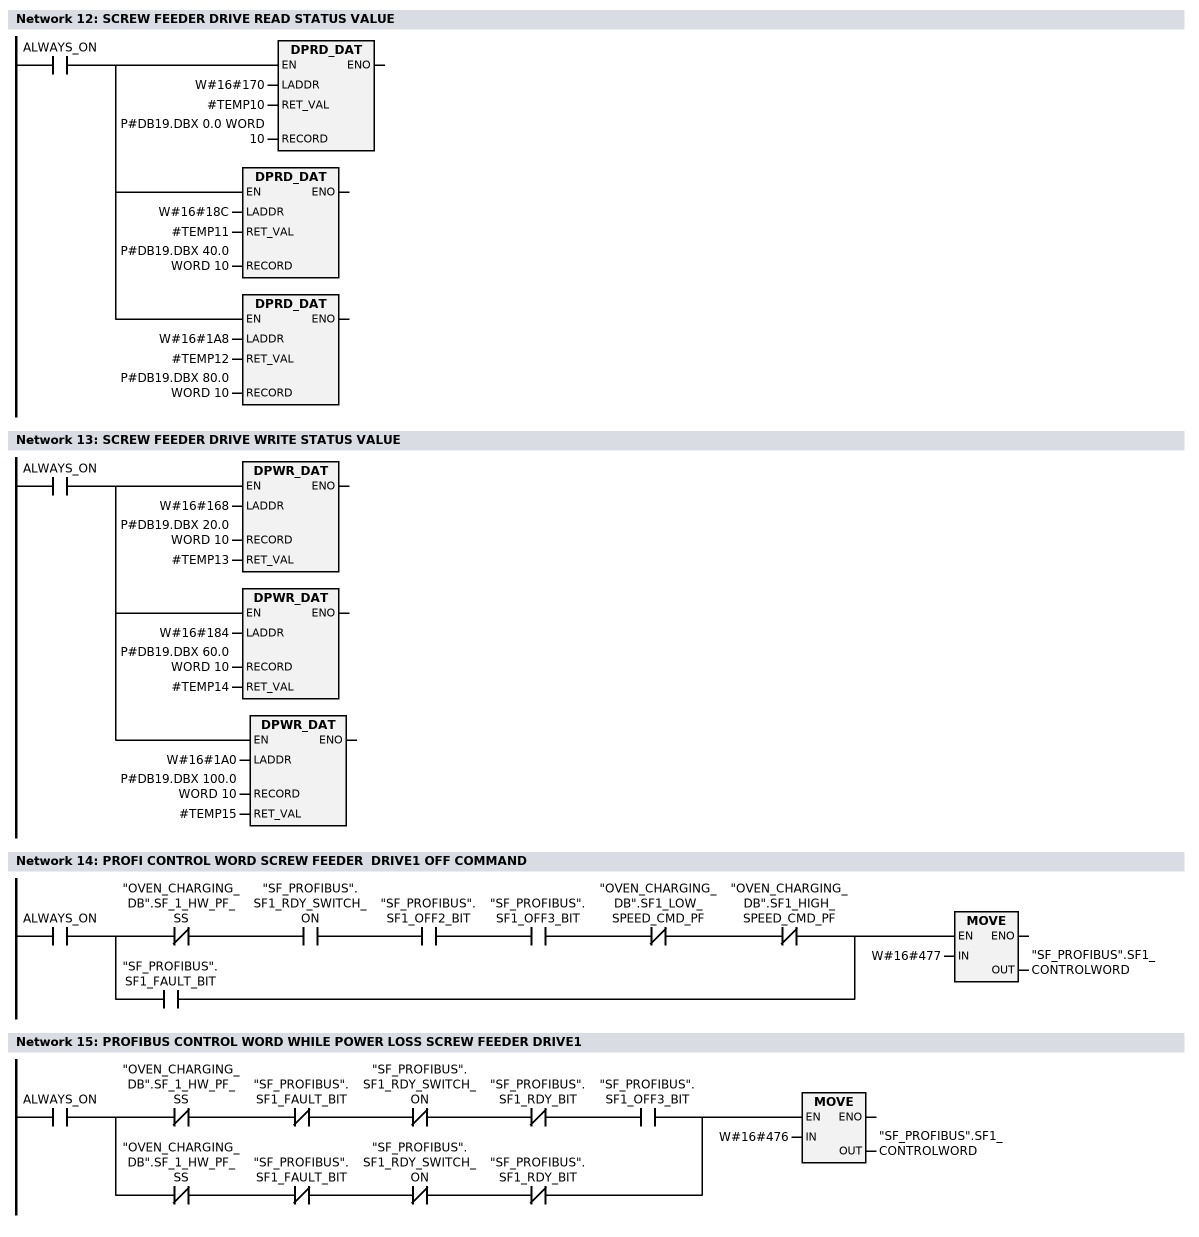
[picture p144: PROFIBUS COMMUNICATION networks 12-15]
NETWORK
TITLE = SCREW FEEDER DRIVE READ STATUS VALUE
      A     "ALWAYS_ON";
      =     L 36.0;
      A     L 36.0;
      JNB   _010;
      CALL  "DPRD_DAT" (
           LADDR                    := W#16#170,
           RET_VAL                  := #TEMP10,
           RECORD                   := P#DB19.DBX 0.0 WORD 10);
_010: NOP   0;
      A     L 36.0;
      JNB   _011;
      CALL  "DPRD_DAT" (
           LADDR                    := W#16#18C,
           RET_VAL                  := #TEMP11,
           RECORD                   := P#DB19.DBX 40.0 WORD 10);
_011: NOP   0;
      A     L 36.0;
      JNB   _012;
      CALL  "DPRD_DAT" (
           LADDR                    := W#16#1A8,
           RET_VAL                  := #TEMP12,
           RECORD                   := P#DB19.DBX 80.0 WORD 10);
_012: NOP   0;
NETWORK
TITLE = SCREW FEEDER DRIVE WRITE STATUS VALUE
      A     "ALWAYS_ON";
      =     L 36.0;
      A     L 36.0;
      JNB   _013;
      CALL  "DPWR_DAT" (
           LADDR                    := W#16#168,
           RECORD                   := P#DB19.DBX 20.0 WORD 10,
           RET_VAL                  := #TEMP13);
_013: NOP   0;
      A     L 36.0;
      JNB   _014;
      CALL  "DPWR_DAT" (
           LADDR                    := W#16#184,
           RECORD                   := P#DB19.DBX 60.0 WORD 10,
           RET_VAL                  := #TEMP14);
_014: NOP   0;
      A     L 36.0;
      JNB   _015;
      CALL  "DPWR_DAT" (
           LADDR                    := W#16#1A0,
           RECORD                   := P#DB19.DBX 100.0 WORD 10,
           RET_VAL                  := #TEMP15);
_015: NOP   0;
NETWORK
TITLE = PROFI CONTROL WORD SCREW FEEDER  DRIVE1 OFF COMMAND
      A     "ALWAYS_ON";
      A(;
      AN    "OVEN_CHARGING_DB".SF_1_HW_PF_SS;
      A     "SF_PROFIBUS".SF1_RDY_SWITCH_ON;
      A     "SF_PROFIBUS".SF1_OFF2_BIT;
      A     "SF_PROFIBUS".SF1_OFF3_BIT;
      AN    "OVEN_CHARGING_DB".SF1_LOW_SPEED_CMD_PF;
      AN    "OVEN_CHARGING_DB".SF1_HIGH_SPEED_CMD_PF;
      O     "SF_PROFIBUS".SF1_FAULT_BIT;
      );
      JNB   _016;
      L     W#16#477;
      T     "SF_PROFIBUS".SF1_CONTROLWORD;
_016: NOP   0;
NETWORK
TITLE = PROFIBUS CONTROL WORD WHILE POWER LOSS SCREW FEEDER DRIVE1
      A     "ALWAYS_ON";
      A(;
      AN    "OVEN_CHARGING_DB".SF_1_HW_PF_SS;
      AN    "SF_PROFIBUS".SF1_FAULT_BIT;
      AN    "SF_PROFIBUS".SF1_RDY_SWITCH_ON;
      AN    "SF_PROFIBUS".SF1_RDY_BIT;
      A     "SF_PROFIBUS".SF1_OFF3_BIT;
      O;
      AN    "OVEN_CHARGING_DB".SF_1_HW_PF_SS;
      AN    "SF_PROFIBUS".SF1_FAULT_BIT;
      AN    "SF_PROFIBUS".SF1_RDY_SWITCH_ON;
      AN    "SF_PROFIBUS".SF1_RDY_BIT;
      );
      JNB   _017;
      L     W#16#476;
      T     "SF_PROFIBUS".SF1_CONTROLWORD;
_017: NOP   0;
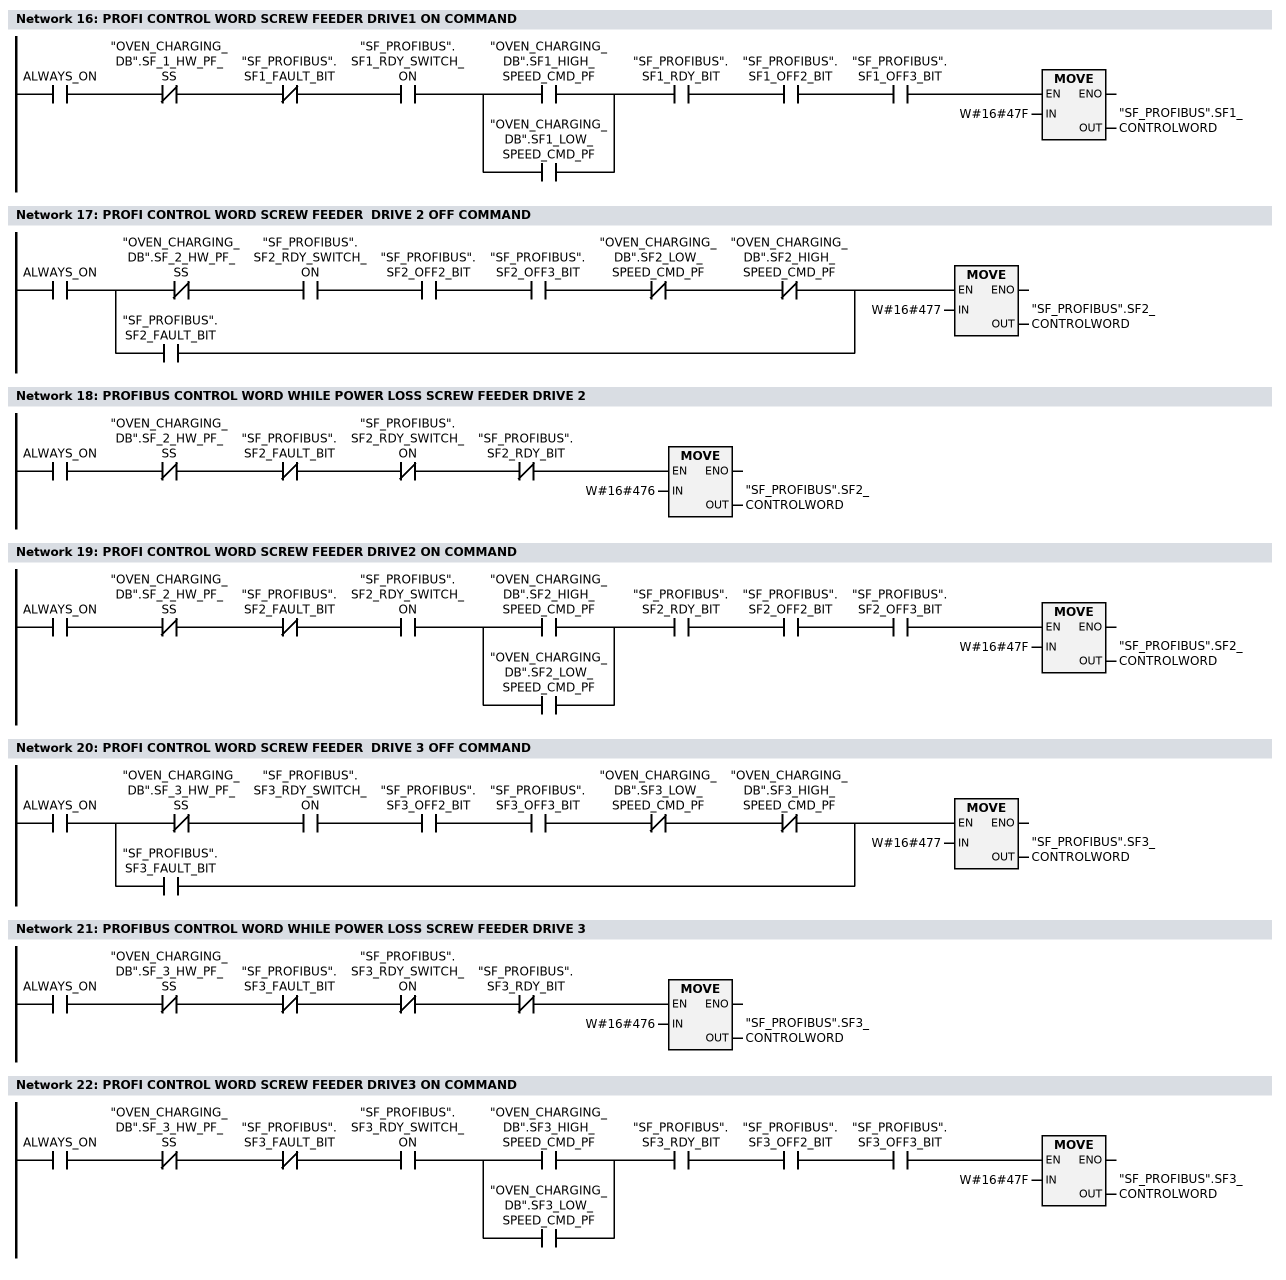
NETWORK
TITLE = PROFI CONTROL WORD SCREW FEEDER DRIVE1 ON COMMAND
      A     "ALWAYS_ON";
      AN    "OVEN_CHARGING_DB".SF_1_HW_PF_SS;
      AN    "SF_PROFIBUS".SF1_FAULT_BIT;
      A     "SF_PROFIBUS".SF1_RDY_SWITCH_ON;
      A(;
      O     "OVEN_CHARGING_DB".SF1_HIGH_SPEED_CMD_PF;
      O     "OVEN_CHARGING_DB".SF1_LOW_SPEED_CMD_PF;
      );
      A     "SF_PROFIBUS".SF1_RDY_BIT;
      A     "SF_PROFIBUS".SF1_OFF2_BIT;
      A     "SF_PROFIBUS".SF1_OFF3_BIT;
      JNB   _018;
      L     W#16#47F;
      T     "SF_PROFIBUS".SF1_CONTROLWORD;
_018: NOP   0;
NETWORK
TITLE = PROFI CONTROL WORD SCREW FEEDER  DRIVE 2 OFF COMMAND
      A     "ALWAYS_ON";
      A(;
      AN    "OVEN_CHARGING_DB".SF_2_HW_PF_SS;
      A     "SF_PROFIBUS".SF2_RDY_SWITCH_ON;
      A     "SF_PROFIBUS".SF2_OFF2_BIT;
      A     "SF_PROFIBUS".SF2_OFF3_BIT;
      AN    "OVEN_CHARGING_DB".SF2_LOW_SPEED_CMD_PF;
      AN    "OVEN_CHARGING_DB".SF2_HIGH_SPEED_CMD_PF;
      O     "SF_PROFIBUS".SF2_FAULT_BIT;
      );
      JNB   _019;
      L     W#16#477;
      T     "SF_PROFIBUS".SF2_CONTROLWORD;
_019: NOP   0;
NETWORK
TITLE = PROFIBUS CONTROL WORD WHILE POWER LOSS SCREW FEEDER DRIVE 2
      A     "ALWAYS_ON";
      AN    "OVEN_CHARGING_DB".SF_2_HW_PF_SS;
      AN    "SF_PROFIBUS".SF2_FAULT_BIT;
      AN    "SF_PROFIBUS".SF2_RDY_SWITCH_ON;
      AN    "SF_PROFIBUS".SF2_RDY_BIT;
      JNB   _01a;
      L     W#16#476;
      T     "SF_PROFIBUS".SF2_CONTROLWORD;
_01a: NOP   0;
NETWORK
TITLE = PROFI CONTROL WORD SCREW FEEDER DRIVE2 ON COMMAND
      A     "ALWAYS_ON";
      AN    "OVEN_CHARGING_DB".SF_2_HW_PF_SS;
      AN    "SF_PROFIBUS".SF2_FAULT_BIT;
      A     "SF_PROFIBUS".SF2_RDY_SWITCH_ON;
      A(;
      O     "OVEN_CHARGING_DB".SF2_HIGH_SPEED_CMD_PF;
      O     "OVEN_CHARGING_DB".SF2_LOW_SPEED_CMD_PF;
      );
      A     "SF_PROFIBUS".SF2_RDY_BIT;
      A     "SF_PROFIBUS".SF2_OFF2_BIT;
      A     "SF_PROFIBUS".SF2_OFF3_BIT;
      JNB   _01b;
      L     W#16#47F;
      T     "SF_PROFIBUS".SF2_CONTROLWORD;
_01b: NOP   0;
NETWORK
TITLE = PROFI CONTROL WORD SCREW FEEDER  DRIVE 3 OFF COMMAND
      A     "ALWAYS_ON";
      A(;
      AN    "OVEN_CHARGING_DB".SF_3_HW_PF_SS;
      A     "SF_PROFIBUS".SF3_RDY_SWITCH_ON;
      A     "SF_PROFIBUS".SF3_OFF2_BIT;
      A     "SF_PROFIBUS".SF3_OFF3_BIT;
      AN    "OVEN_CHARGING_DB".SF3_LOW_SPEED_CMD_PF;
      AN    "OVEN_CHARGING_DB".SF3_HIGH_SPEED_CMD_PF;
      O     "SF_PROFIBUS".SF3_FAULT_BIT;
      );
      JNB   _01c;
      L     W#16#477;
      T     "SF_PROFIBUS".SF3_CONTROLWORD;
_01c: NOP   0;
NETWORK
TITLE = PROFIBUS CONTROL WORD WHILE POWER LOSS SCREW FEEDER DRIVE 3
      A     "ALWAYS_ON";
      AN    "OVEN_CHARGING_DB".SF_3_HW_PF_SS;
      AN    "SF_PROFIBUS".SF3_FAULT_BIT;
      AN    "SF_PROFIBUS".SF3_RDY_SWITCH_ON;
      AN    "SF_PROFIBUS".SF3_RDY_BIT;
      JNB   _01d;
      L     W#16#476;
      T     "SF_PROFIBUS".SF3_CONTROLWORD;
_01d: NOP   0;
NETWORK
TITLE = PROFI CONTROL WORD SCREW FEEDER DRIVE3 ON COMMAND
      A     "ALWAYS_ON";
      AN    "OVEN_CHARGING_DB".SF_3_HW_PF_SS;
      AN    "SF_PROFIBUS".SF3_FAULT_BIT;
      A     "SF_PROFIBUS".SF3_RDY_SWITCH_ON;
      A(;
      O     "OVEN_CHARGING_DB".SF3_HIGH_SPEED_CMD_PF;
      O     "OVEN_CHARGING_DB".SF3_LOW_SPEED_CMD_PF;
      );
      A     "SF_PROFIBUS".SF3_RDY_BIT;
      A     "SF_PROFIBUS".SF3_OFF2_BIT;
      A     "SF_PROFIBUS".SF3_OFF3_BIT;
      JNB   _01e;
      L     W#16#47F;
      T     "SF_PROFIBUS".SF3_CONTROLWORD;
_01e: NOP   0;
END_FUNCTION

FUNCTION "LID_2_MECHANISM" : VOID	// FC 13
//AUTO SEQ
//Prepare to charge pb 
//Carriage Fwd 
//Vert Down 
//Mag On
//Osc On
//3s 
//Osc off
//Lid at mag
//Ver Up
//Car Ret 
//// Frm clnr down if bypass
//Car fwd 
//car Ver cln pos down 
//Frm clnr Mtr on 
//5s 
//off 
//car Ver  up 
//Car Ret //
//Teles Down 
AUTHOR : Arun
VERSION : 0.1
BEGIN
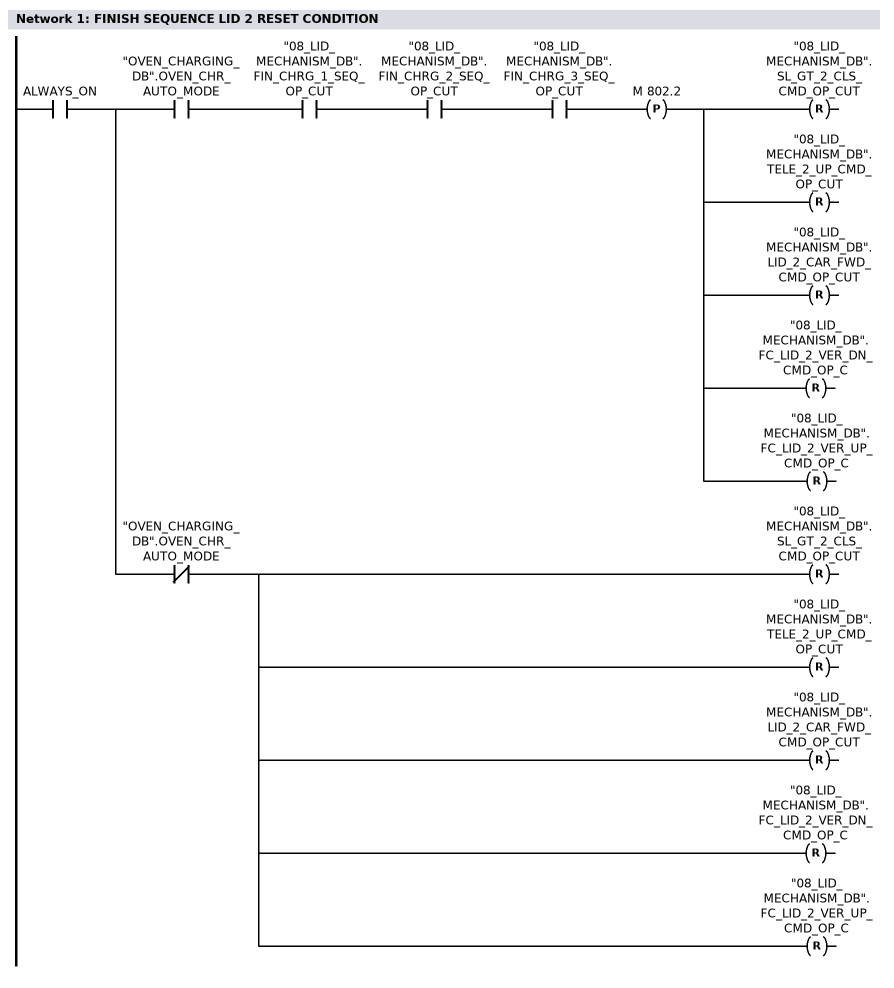
NETWORK
TITLE = FINISH SEQUENCE LID 2 RESET CONDITION
      A     "ALWAYS_ON";
      =     L 0.0;
      A     L 0.0;
      A     "OVEN_CHARGING_DB".OVEN_CHR_AUTO_MODE;
      A     "08_LID_MECHANISM_DB".FIN_CHRG_1_SEQ_OP_CUT;
      A     "08_LID_MECHANISM_DB".FIN_CHRG_2_SEQ_OP_CUT;
      A     "08_LID_MECHANISM_DB".FIN_CHRG_3_SEQ_OP_CUT;
      FP    M 802.2;
      R     "08_LID_MECHANISM_DB".SL_GT_2_CLS_CMD_OP_CUT;
      R     "08_LID_MECHANISM_DB".TELE_2_UP_CMD_OP_CUT;
      R     "08_LID_MECHANISM_DB".LID_2_CAR_FWD_CMD_OP_CUT;
      R     "08_LID_MECHANISM_DB".FC_LID_2_VER_DN_CMD_OP_C;
      R     "08_LID_MECHANISM_DB".FC_LID_2_VER_UP_CMD_OP_C;
      A     L 0.0;
      AN    "OVEN_CHARGING_DB".OVEN_CHR_AUTO_MODE;
      R     "08_LID_MECHANISM_DB".SL_GT_2_CLS_CMD_OP_CUT;
      R     "08_LID_MECHANISM_DB".TELE_2_UP_CMD_OP_CUT;
      R     "08_LID_MECHANISM_DB".LID_2_CAR_FWD_CMD_OP_CUT;
      R     "08_LID_MECHANISM_DB".FC_LID_2_VER_DN_CMD_OP_C;
      R     "08_LID_MECHANISM_DB".FC_LID_2_VER_UP_CMD_OP_C;
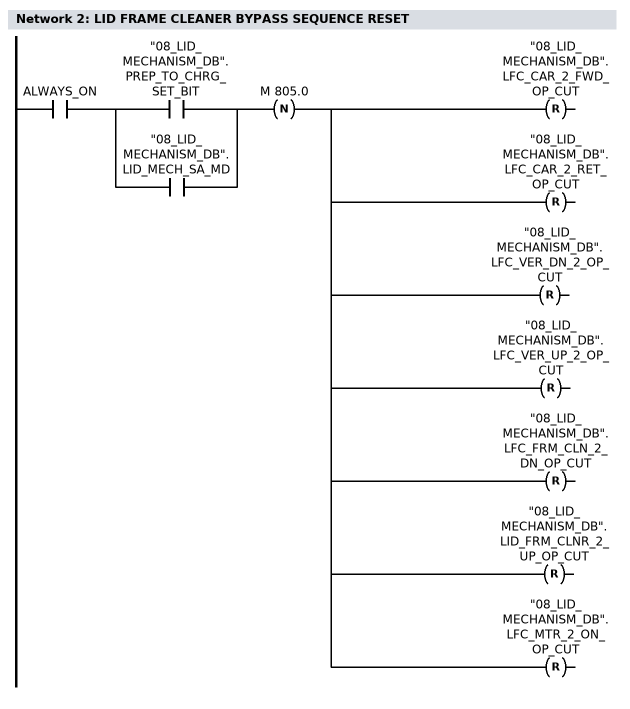
NETWORK
TITLE = LID FRAME CLEANER BYPASS SEQUENCE RESET
      A     "ALWAYS_ON";
      A(;
      O     "08_LID_MECHANISM_DB".PREP_TO_CHRG_SET_BIT;
      O     "08_LID_MECHANISM_DB".LID_MECH_SA_MD;
      );
      FN    M 805.0;
      R     "08_LID_MECHANISM_DB".LFC_CAR_2_FWD_OP_CUT;
      R     "08_LID_MECHANISM_DB".LFC_CAR_2_RET_OP_CUT;
      R     "08_LID_MECHANISM_DB".LFC_VER_DN_2_OP_CUT;
      R     "08_LID_MECHANISM_DB".LFC_VER_UP_2_OP_CUT;
      R     "08_LID_MECHANISM_DB".LFC_FRM_CLN_2_DN_OP_CUT;
      R     "08_LID_MECHANISM_DB".LID_FRM_CLNR_2_UP_OP_CUT;
      R     "08_LID_MECHANISM_DB".LFC_MTR_2_ON_OP_CUT;
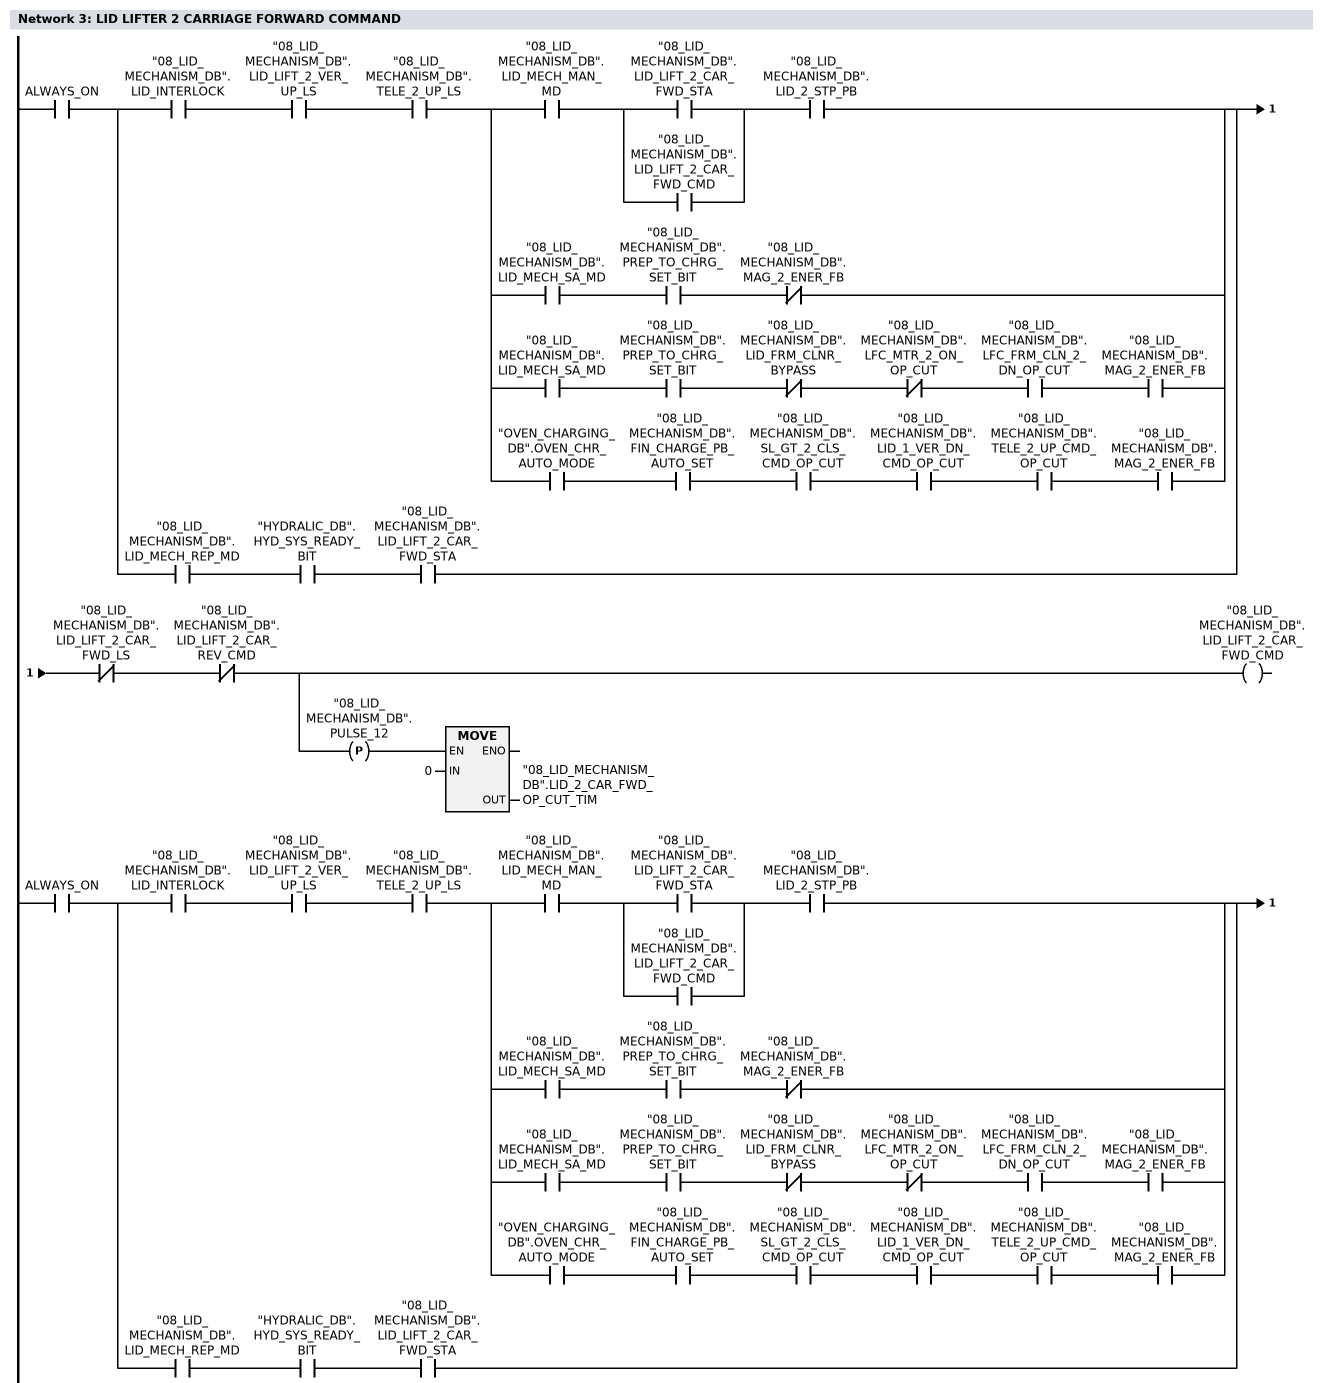
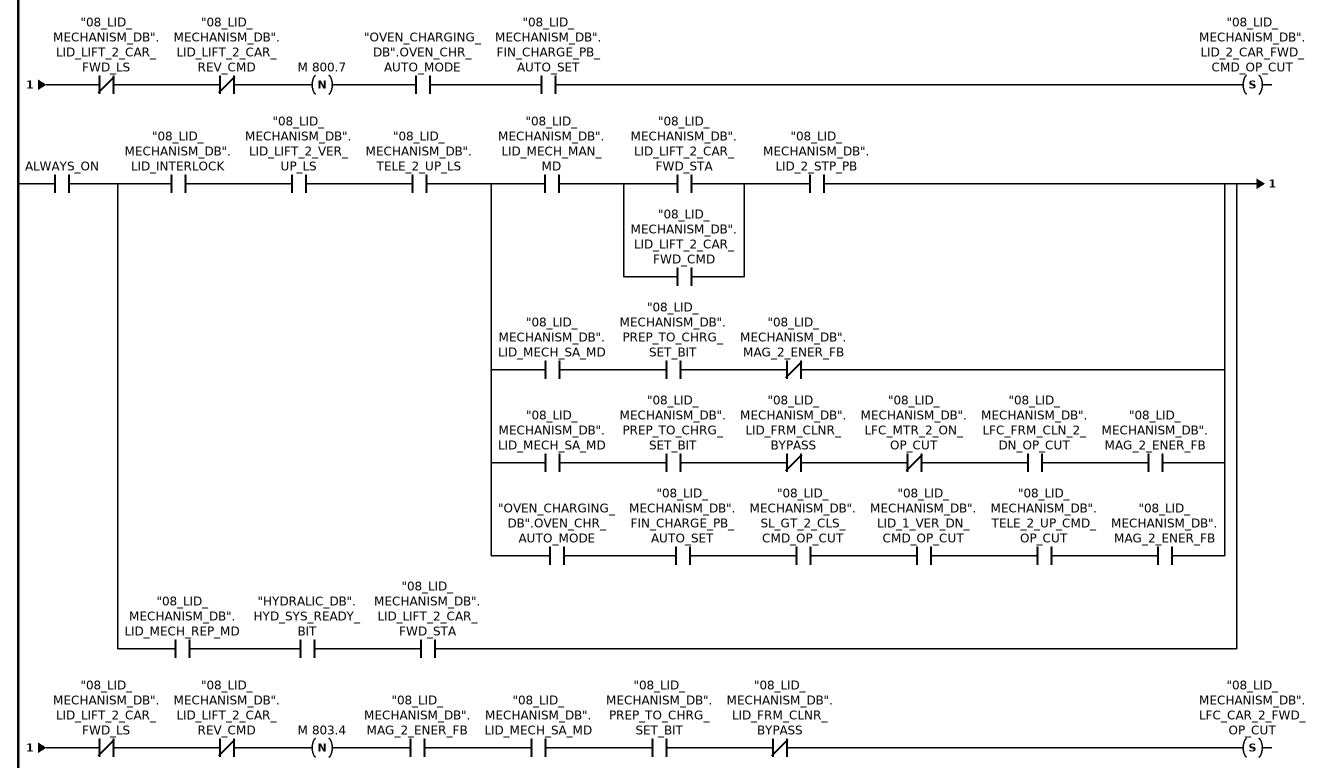
NETWORK
TITLE = LID LIFTER 2 CARRIAGE FORWARD COMMAND
      A     "ALWAYS_ON";
      A(;
      A     "08_LID_MECHANISM_DB".LID_INTERLOCK;
      A     "08_LID_MECHANISM_DB".LID_LIFT_2_VER_UP_LS;
      A     "08_LID_MECHANISM_DB".TELE_2_UP_LS;
      A(;
      A     "08_LID_MECHANISM_DB".LID_MECH_MAN_MD;
      A(;
      O     "08_LID_MECHANISM_DB".LID_LIFT_2_CAR_FWD_STA;
      O     "08_LID_MECHANISM_DB".LID_LIFT_2_CAR_FWD_CMD;
      );
      A     "08_LID_MECHANISM_DB".LID_2_STP_PB;
      O;
      A     "08_LID_MECHANISM_DB".LID_MECH_SA_MD;
      A     "08_LID_MECHANISM_DB".PREP_TO_CHRG_SET_BIT;
      AN    "08_LID_MECHANISM_DB".MAG_2_ENER_FB;
      O;
      A     "08_LID_MECHANISM_DB".LID_MECH_SA_MD;
      A     "08_LID_MECHANISM_DB".PREP_TO_CHRG_SET_BIT;
      AN    "08_LID_MECHANISM_DB".LID_FRM_CLNR_BYPASS;
      AN    "08_LID_MECHANISM_DB".LFC_MTR_2_ON_OP_CUT;
      A     "08_LID_MECHANISM_DB".LFC_FRM_CLN_2_DN_OP_CUT;
      A     "08_LID_MECHANISM_DB".MAG_2_ENER_FB;
      O;
      A     "OVEN_CHARGING_DB".OVEN_CHR_AUTO_MODE;
      A     "08_LID_MECHANISM_DB".FIN_CHARGE_PB_AUTO_SET;
      A     "08_LID_MECHANISM_DB".SL_GT_2_CLS_CMD_OP_CUT;
      A     "08_LID_MECHANISM_DB".LID_1_VER_DN_CMD_OP_CUT;
      A     "08_LID_MECHANISM_DB".TELE_2_UP_CMD_OP_CUT;
      A     "08_LID_MECHANISM_DB".MAG_2_ENER_FB;
      );
      O;
      A     "08_LID_MECHANISM_DB".LID_MECH_REP_MD;
      A     "HYDRALIC_DB".HYD_SYS_READY_BIT;
      A     "08_LID_MECHANISM_DB".LID_LIFT_2_CAR_FWD_STA;
      );
      AN    "08_LID_MECHANISM_DB".LID_LIFT_2_CAR_FWD_LS;
      AN    "08_LID_MECHANISM_DB".LID_LIFT_2_CAR_REV_CMD;
      =     L 0.0;
      A     L 0.0;
      BLD   102;
      =     "08_LID_MECHANISM_DB".LID_LIFT_2_CAR_FWD_CMD;
      A     L 0.0;
      FP    "08_LID_MECHANISM_DB".PULSE_12;
      JNB   _001;
      L     0;
      T     "08_LID_MECHANISM_DB".LID_2_CAR_FWD_OP_CUT_TIM;
_001: NOP   0;
      A(;
      A     L 0.0;
      FN    M 800.7;
      );
      A     "OVEN_CHARGING_DB".OVEN_CHR_AUTO_MODE;
      A     "08_LID_MECHANISM_DB".FIN_CHARGE_PB_AUTO_SET;
      S     "08_LID_MECHANISM_DB".LID_2_CAR_FWD_CMD_OP_CUT;
      A(;
      A     L 0.0;
      FN    M 803.4;
      );
      A     "08_LID_MECHANISM_DB".MAG_2_ENER_FB;
      A     "08_LID_MECHANISM_DB".LID_MECH_SA_MD;
      A     "08_LID_MECHANISM_DB".PREP_TO_CHRG_SET_BIT;
      AN    "08_LID_MECHANISM_DB".LID_FRM_CLNR_BYPASS;
      S     "08_LID_MECHANISM_DB".LFC_CAR_2_FWD_OP_CUT;
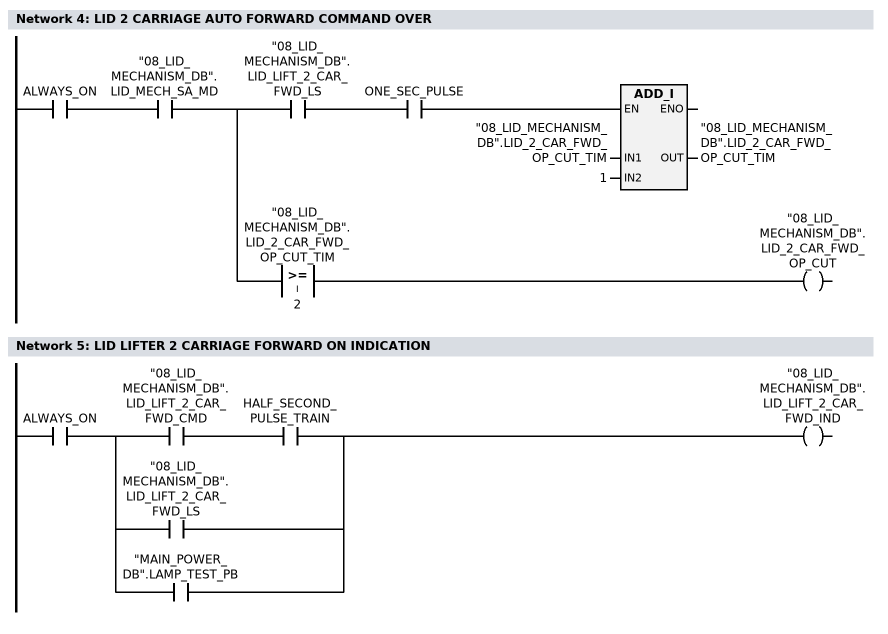
NETWORK
TITLE = LID 2 CARRIAGE AUTO FORWARD COMMAND OVER
      A     "ALWAYS_ON";
      A     "08_LID_MECHANISM_DB".LID_MECH_SA_MD;
      =     L 0.0;
      A     L 0.0;
      A     "08_LID_MECHANISM_DB".LID_LIFT_2_CAR_FWD_LS;
      A     "ONE_SEC_PULSE";
      JNB   _002;
      L     "08_LID_MECHANISM_DB".LID_2_CAR_FWD_OP_CUT_TIM;
      L     1;
      +I;
      T     "08_LID_MECHANISM_DB".LID_2_CAR_FWD_OP_CUT_TIM;
_002: NOP   0;
      A     L 0.0;
      A(;
      L     "08_LID_MECHANISM_DB".LID_2_CAR_FWD_OP_CUT_TIM;
      L     2;
      >=I;
      );
      =     "08_LID_MECHANISM_DB".LID_2_CAR_FWD_OP_CUT;
NETWORK
TITLE = LID LIFTER 2 CARRIAGE FORWARD ON INDICATION
      A     "ALWAYS_ON";
      A(;
      A     "08_LID_MECHANISM_DB".LID_LIFT_2_CAR_FWD_CMD;
      A     "HALF_SECOND_PULSE_TRAIN";
      O     "08_LID_MECHANISM_DB".LID_LIFT_2_CAR_FWD_LS;
      O     "MAIN_POWER_DB".LAMP_TEST_PB;
      );
      =     "08_LID_MECHANISM_DB".LID_LIFT_2_CAR_FWD_IND;
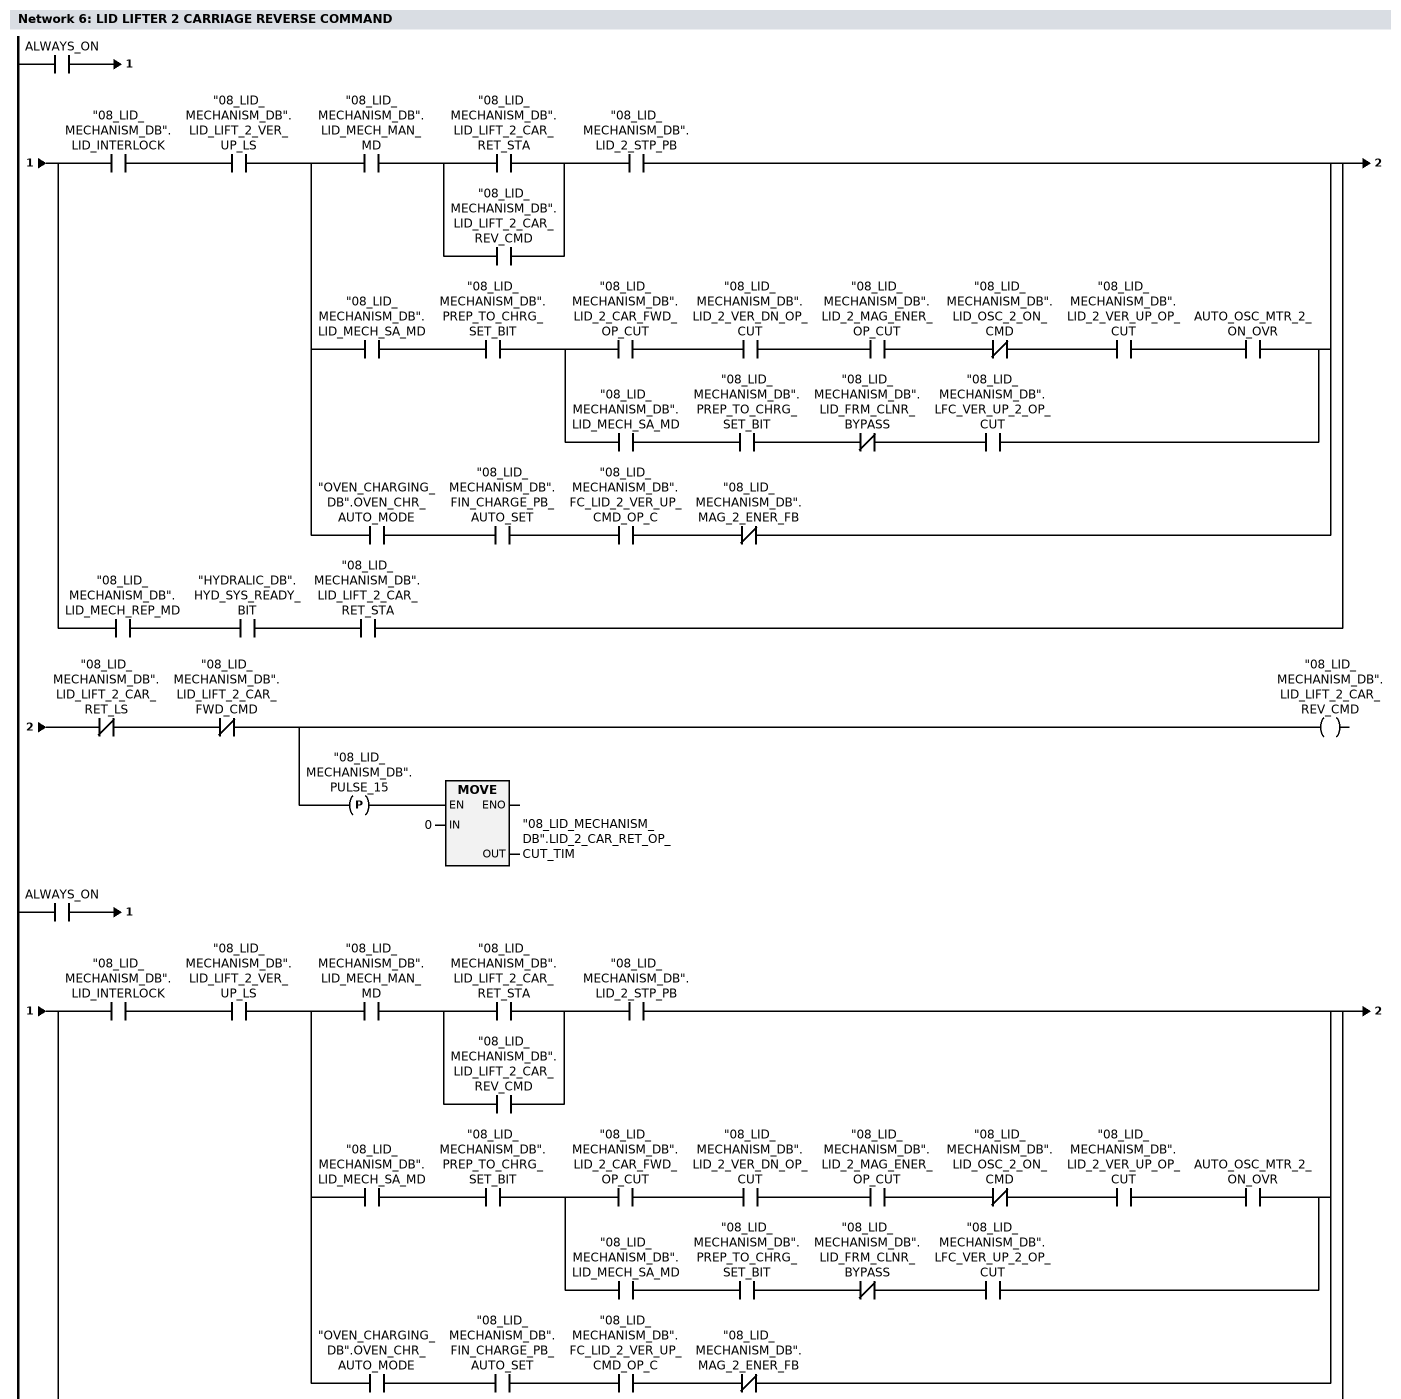
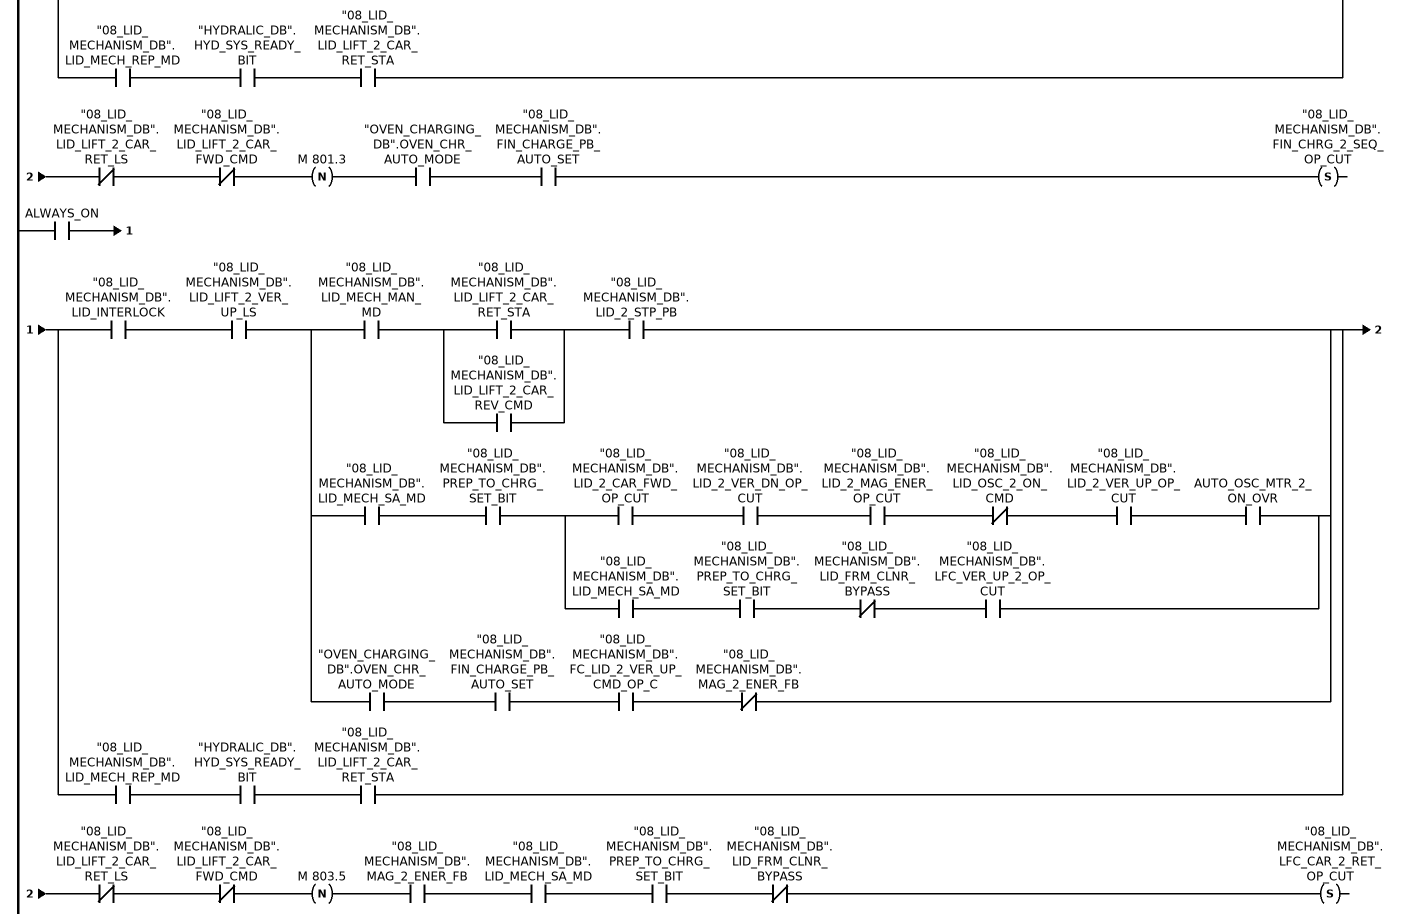
NETWORK
TITLE = LID LIFTER 2 CARRIAGE REVERSE COMMAND
      A     "ALWAYS_ON";
      A(;
      A     "08_LID_MECHANISM_DB".LID_INTERLOCK;
      A     "08_LID_MECHANISM_DB".LID_LIFT_2_VER_UP_LS;
      A(;
      A     "08_LID_MECHANISM_DB".LID_MECH_MAN_MD;
      A(;
      O     "08_LID_MECHANISM_DB".LID_LIFT_2_CAR_RET_STA;
      O     "08_LID_MECHANISM_DB".LID_LIFT_2_CAR_REV_CMD;
      );
      A     "08_LID_MECHANISM_DB".LID_2_STP_PB;
      O;
      A     "08_LID_MECHANISM_DB".LID_MECH_SA_MD;
      A     "08_LID_MECHANISM_DB".PREP_TO_CHRG_SET_BIT;
      A(;
      A     "08_LID_MECHANISM_DB".LID_2_CAR_FWD_OP_CUT;
      A     "08_LID_MECHANISM_DB".LID_2_VER_DN_OP_CUT;
      A     "08_LID_MECHANISM_DB".LID_2_MAG_ENER_OP_CUT;
      AN    "08_LID_MECHANISM_DB".LID_OSC_2_ON_CMD;
      A     "08_LID_MECHANISM_DB".LID_2_VER_UP_OP_CUT;
      A     "AUTO_OSC_MTR_2_ON_OVR";
      O;
      A     "08_LID_MECHANISM_DB".LID_MECH_SA_MD;
      A     "08_LID_MECHANISM_DB".PREP_TO_CHRG_SET_BIT;
      AN    "08_LID_MECHANISM_DB".LID_FRM_CLNR_BYPASS;
      A     "08_LID_MECHANISM_DB".LFC_VER_UP_2_OP_CUT;
      );
      O;
      A     "OVEN_CHARGING_DB".OVEN_CHR_AUTO_MODE;
      A     "08_LID_MECHANISM_DB".FIN_CHARGE_PB_AUTO_SET;
      A     "08_LID_MECHANISM_DB".FC_LID_2_VER_UP_CMD_OP_C;
      AN    "08_LID_MECHANISM_DB".MAG_2_ENER_FB;
      );
      O;
      A     "08_LID_MECHANISM_DB".LID_MECH_REP_MD;
      A     "HYDRALIC_DB".HYD_SYS_READY_BIT;
      A     "08_LID_MECHANISM_DB".LID_LIFT_2_CAR_RET_STA;
      );
      AN    "08_LID_MECHANISM_DB".LID_LIFT_2_CAR_RET_LS;
      AN    "08_LID_MECHANISM_DB".LID_LIFT_2_CAR_FWD_CMD;
      =     L 0.0;
      A     L 0.0;
      BLD   102;
      =     "08_LID_MECHANISM_DB".LID_LIFT_2_CAR_REV_CMD;
      A     L 0.0;
      FP    "08_LID_MECHANISM_DB".PULSE_15;
      JNB   _003;
      L     0;
      T     "08_LID_MECHANISM_DB".LID_2_CAR_RET_OP_CUT_TIM;
_003: NOP   0;
      A(;
      A     L 0.0;
      FN    M 801.3;
      );
      A     "OVEN_CHARGING_DB".OVEN_CHR_AUTO_MODE;
      A     "08_LID_MECHANISM_DB".FIN_CHARGE_PB_AUTO_SET;
      S     "08_LID_MECHANISM_DB".FIN_CHRG_2_SEQ_OP_CUT;
      A(;
      A     L 0.0;
      FN    M 803.5;
      );
      A     "08_LID_MECHANISM_DB".MAG_2_ENER_FB;
      A     "08_LID_MECHANISM_DB".LID_MECH_SA_MD;
      A     "08_LID_MECHANISM_DB".PREP_TO_CHRG_SET_BIT;
      AN    "08_LID_MECHANISM_DB".LID_FRM_CLNR_BYPASS;
      S     "08_LID_MECHANISM_DB".LFC_CAR_2_RET_OP_CUT;
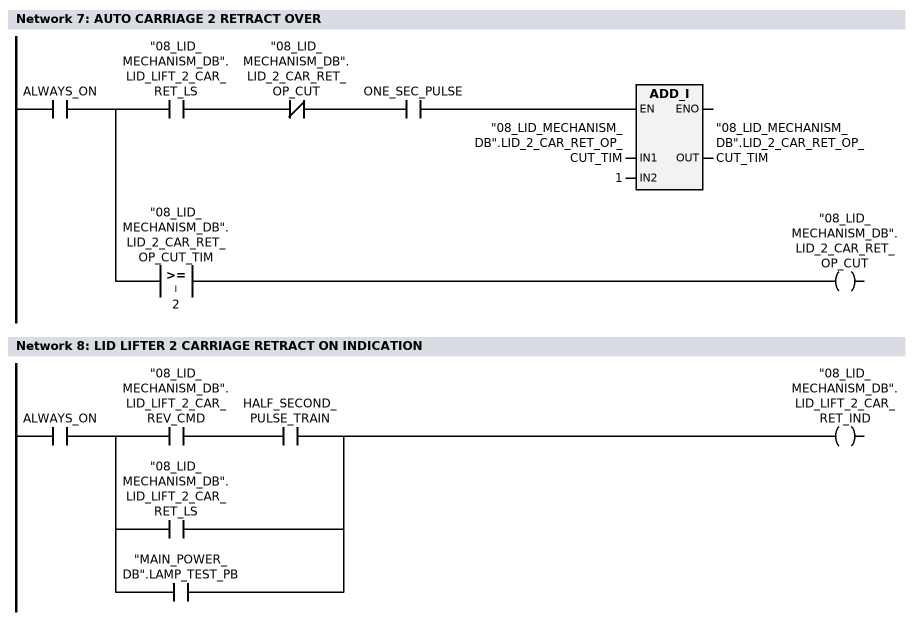
NETWORK
TITLE = AUTO CARRIAGE 2 RETRACT OVER
      A     "ALWAYS_ON";
      =     L 0.0;
      A     L 0.0;
      A     "08_LID_MECHANISM_DB".LID_LIFT_2_CAR_RET_LS;
      AN    "08_LID_MECHANISM_DB".LID_2_CAR_RET_OP_CUT;
      A     "ONE_SEC_PULSE";
      JNB   _004;
      L     "08_LID_MECHANISM_DB".LID_2_CAR_RET_OP_CUT_TIM;
      L     1;
      +I;
      T     "08_LID_MECHANISM_DB".LID_2_CAR_RET_OP_CUT_TIM;
_004: NOP   0;
      A     L 0.0;
      A(;
      L     "08_LID_MECHANISM_DB".LID_2_CAR_RET_OP_CUT_TIM;
      L     2;
      >=I;
      );
      =     "08_LID_MECHANISM_DB".LID_2_CAR_RET_OP_CUT;
NETWORK
TITLE = LID LIFTER 2 CARRIAGE RETRACT ON INDICATION
      A     "ALWAYS_ON";
      A(;
      A     "08_LID_MECHANISM_DB".LID_LIFT_2_CAR_REV_CMD;
      A     "HALF_SECOND_PULSE_TRAIN";
      O     "08_LID_MECHANISM_DB".LID_LIFT_2_CAR_RET_LS;
      O     "MAIN_POWER_DB".LAMP_TEST_PB;
      );
      =     "08_LID_MECHANISM_DB".LID_LIFT_2_CAR_RET_IND;
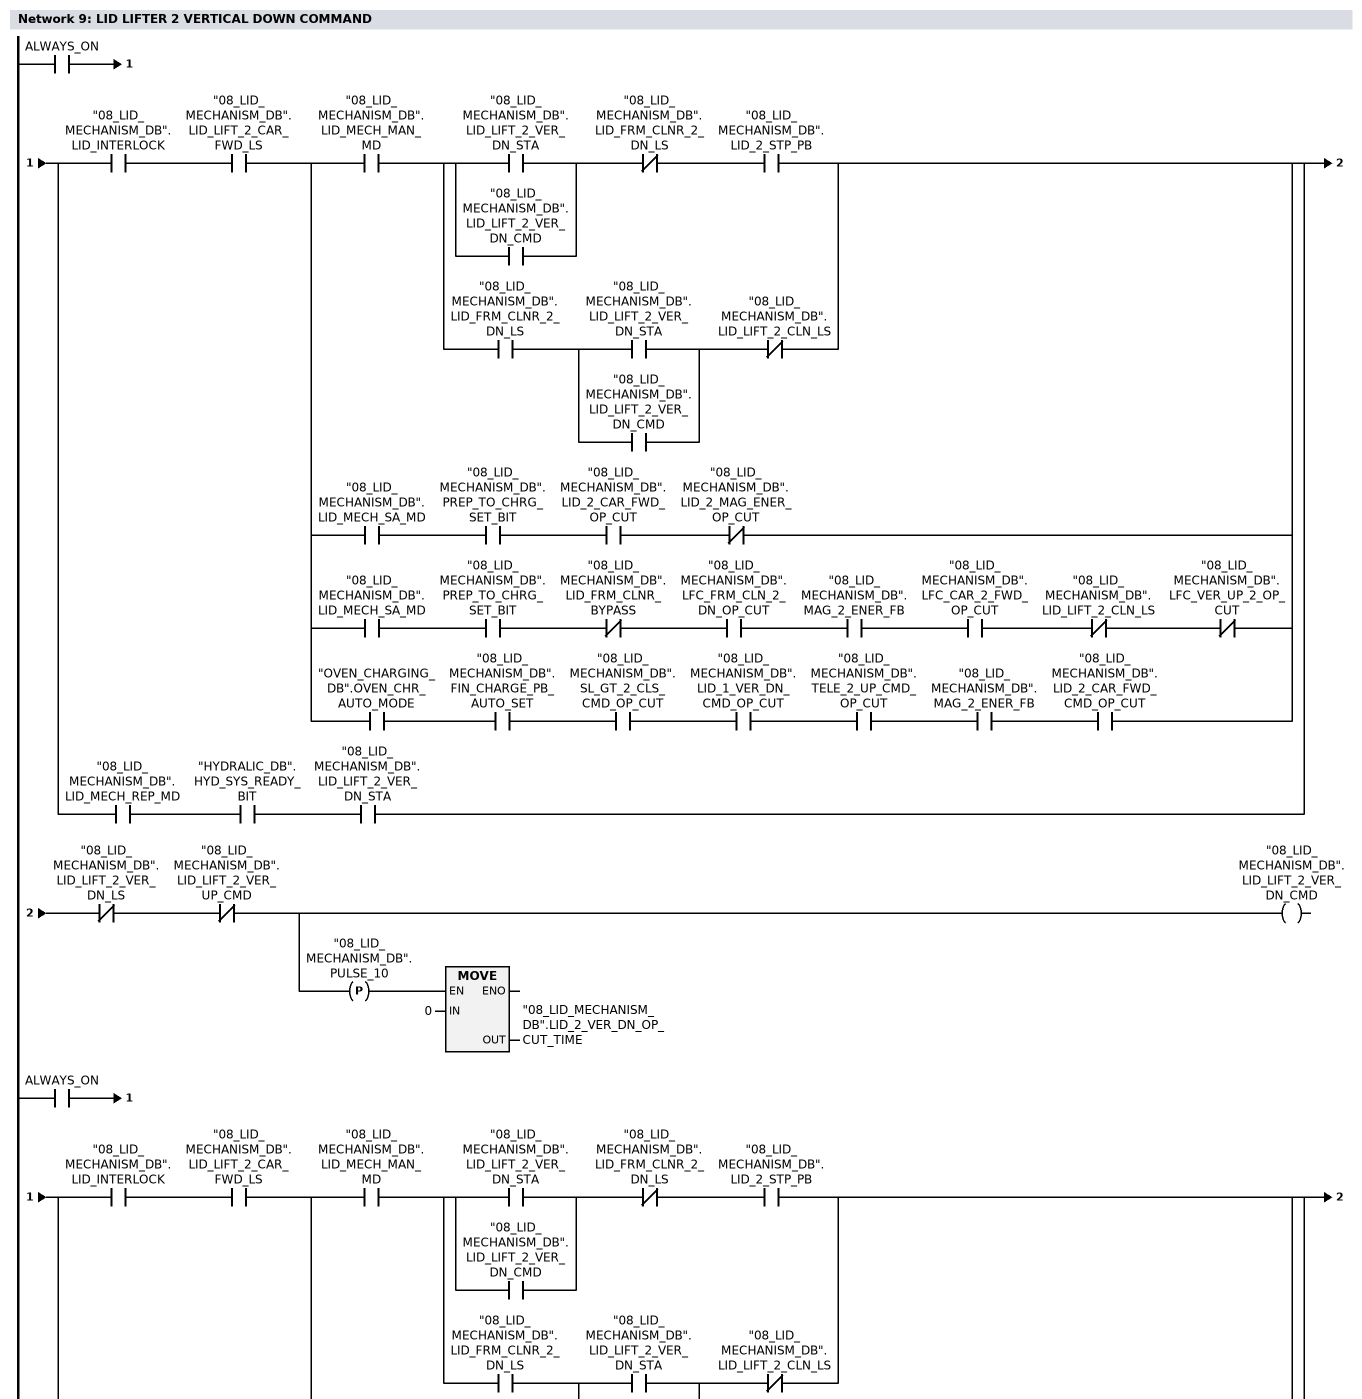
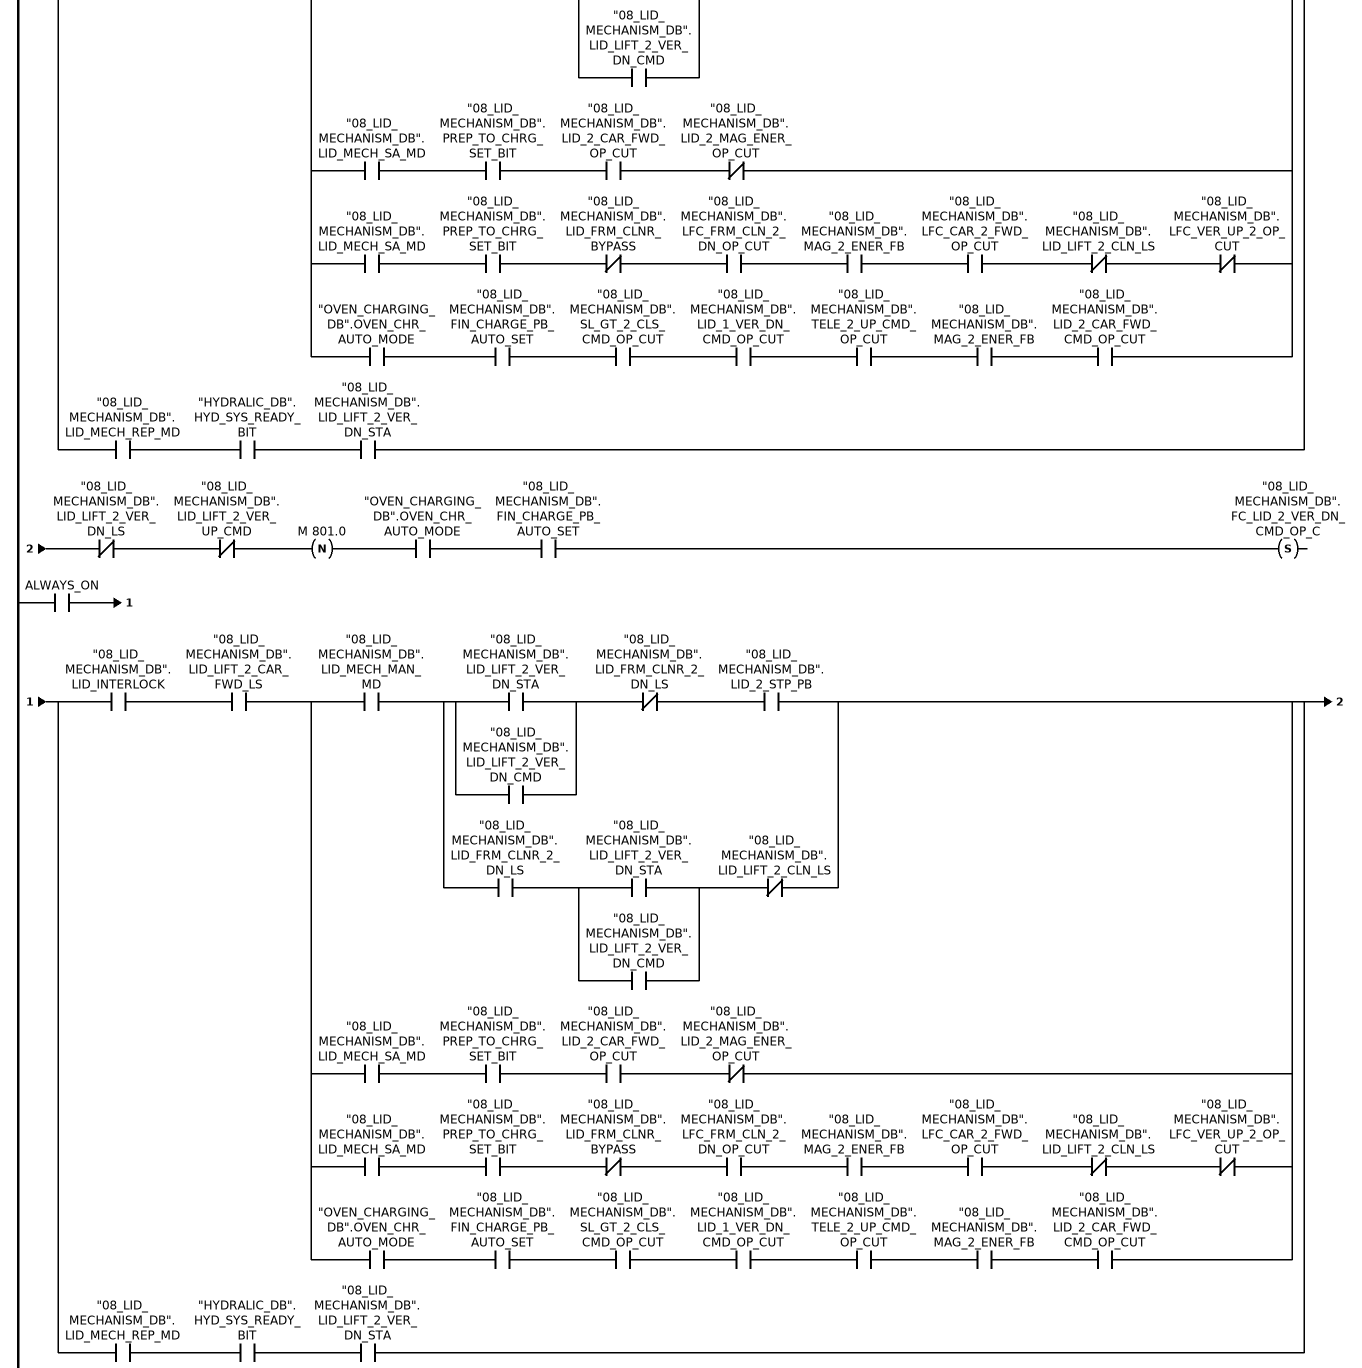
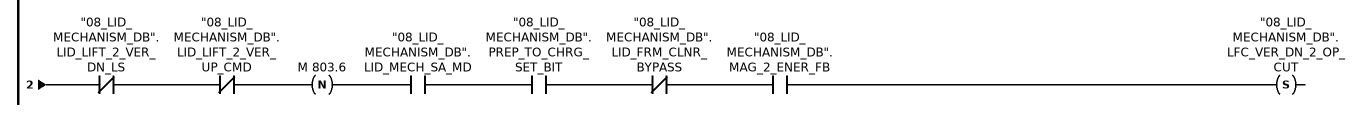
NETWORK
TITLE = LID LIFTER 2 VERTICAL DOWN COMMAND
//PENDING LID FRM BYPASS
//NEXT SEQ .. MAG OFF
      A     "ALWAYS_ON";
      A(;
      A     "08_LID_MECHANISM_DB".LID_INTERLOCK;
      A     "08_LID_MECHANISM_DB".LID_LIFT_2_CAR_FWD_LS;
      A(;
      A     "08_LID_MECHANISM_DB".LID_MECH_MAN_MD;
      A(;
      A(;
      O     "08_LID_MECHANISM_DB".LID_LIFT_2_VER_DN_STA;
      O     "08_LID_MECHANISM_DB".LID_LIFT_2_VER_DN_CMD;
      );
      AN    "08_LID_MECHANISM_DB".LID_FRM_CLNR_2_DN_LS;
      A     "08_LID_MECHANISM_DB".LID_2_STP_PB;
      O;
      A     "08_LID_MECHANISM_DB".LID_FRM_CLNR_2_DN_LS;
      A(;
      O     "08_LID_MECHANISM_DB".LID_LIFT_2_VER_DN_STA;
      O     "08_LID_MECHANISM_DB".LID_LIFT_2_VER_DN_CMD;
      );
      AN    "08_LID_MECHANISM_DB".LID_LIFT_2_CLN_LS;
      );
      O;
      A     "08_LID_MECHANISM_DB".LID_MECH_SA_MD;
      A     "08_LID_MECHANISM_DB".PREP_TO_CHRG_SET_BIT;
      A     "08_LID_MECHANISM_DB".LID_2_CAR_FWD_OP_CUT;
      AN    "08_LID_MECHANISM_DB".LID_2_MAG_ENER_OP_CUT;
      O;
      A     "08_LID_MECHANISM_DB".LID_MECH_SA_MD;
      A     "08_LID_MECHANISM_DB".PREP_TO_CHRG_SET_BIT;
      AN    "08_LID_MECHANISM_DB".LID_FRM_CLNR_BYPASS;
      A     "08_LID_MECHANISM_DB".LFC_FRM_CLN_2_DN_OP_CUT;
      A     "08_LID_MECHANISM_DB".MAG_2_ENER_FB;
      A     "08_LID_MECHANISM_DB".LFC_CAR_2_FWD_OP_CUT;
      AN    "08_LID_MECHANISM_DB".LID_LIFT_2_CLN_LS;
      AN    "08_LID_MECHANISM_DB".LFC_VER_UP_2_OP_CUT;
      O;
      A     "OVEN_CHARGING_DB".OVEN_CHR_AUTO_MODE;
      A     "08_LID_MECHANISM_DB".FIN_CHARGE_PB_AUTO_SET;
      A     "08_LID_MECHANISM_DB".SL_GT_2_CLS_CMD_OP_CUT;
      A     "08_LID_MECHANISM_DB".LID_1_VER_DN_CMD_OP_CUT;
      A     "08_LID_MECHANISM_DB".TELE_2_UP_CMD_OP_CUT;
      A     "08_LID_MECHANISM_DB".MAG_2_ENER_FB;
      A     "08_LID_MECHANISM_DB".LID_2_CAR_FWD_CMD_OP_CUT;
      );
      O;
      A     "08_LID_MECHANISM_DB".LID_MECH_REP_MD;
      A     "HYDRALIC_DB".HYD_SYS_READY_BIT;
      A     "08_LID_MECHANISM_DB".LID_LIFT_2_VER_DN_STA;
      );
      AN    "08_LID_MECHANISM_DB".LID_LIFT_2_VER_DN_LS;
      AN    "08_LID_MECHANISM_DB".LID_LIFT_2_VER_UP_CMD;
      =     L 0.0;
      A     L 0.0;
      BLD   102;
      =     "08_LID_MECHANISM_DB".LID_LIFT_2_VER_DN_CMD;
      A     L 0.0;
      FP    "08_LID_MECHANISM_DB".PULSE_10;
      JNB   _005;
      L     0;
      T     "08_LID_MECHANISM_DB".LID_2_VER_DN_OP_CUT_TIME;
_005: NOP   0;
      A(;
      A     L 0.0;
      FN    M 801.0;
      );
      A     "OVEN_CHARGING_DB".OVEN_CHR_AUTO_MODE;
      A     "08_LID_MECHANISM_DB".FIN_CHARGE_PB_AUTO_SET;
      S     "08_LID_MECHANISM_DB".FC_LID_2_VER_DN_CMD_OP_C;
      A(;
      A     L 0.0;
      FN    M 803.6;
      );
      A     "08_LID_MECHANISM_DB".LID_MECH_SA_MD;
      A     "08_LID_MECHANISM_DB".PREP_TO_CHRG_SET_BIT;
      AN    "08_LID_MECHANISM_DB".LID_FRM_CLNR_BYPASS;
      A     "08_LID_MECHANISM_DB".MAG_2_ENER_FB;
      S     "08_LID_MECHANISM_DB".LFC_VER_DN_2_OP_CUT;
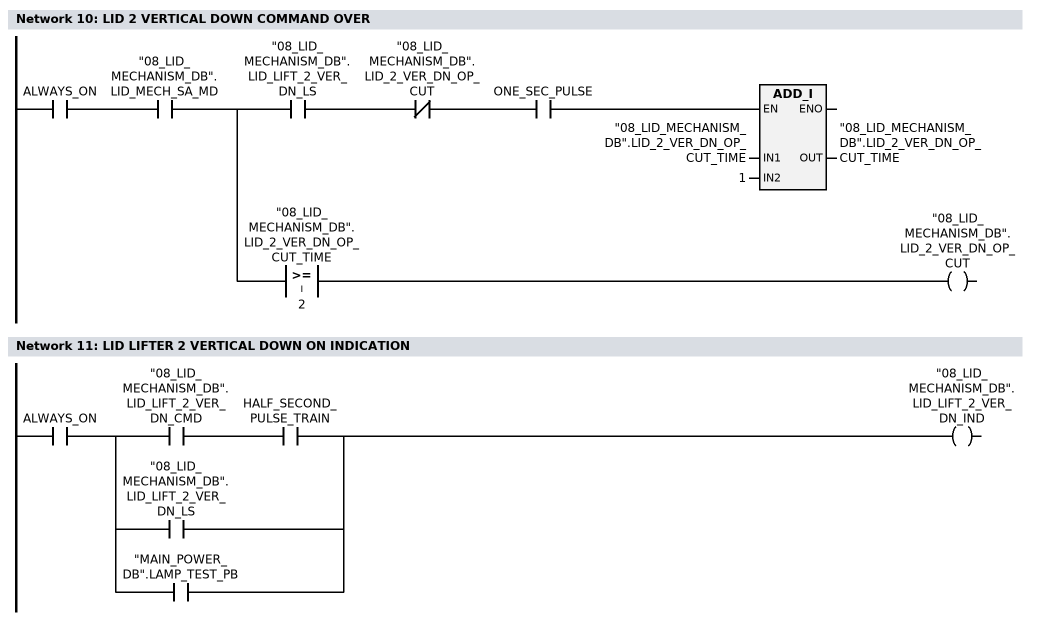
NETWORK
TITLE = LID 2 VERTICAL DOWN COMMAND OVER
      A     "ALWAYS_ON";
      A     "08_LID_MECHANISM_DB".LID_MECH_SA_MD;
      =     L 0.0;
      A     L 0.0;
      A     "08_LID_MECHANISM_DB".LID_LIFT_2_VER_DN_LS;
      AN    "08_LID_MECHANISM_DB".LID_2_VER_DN_OP_CUT;
      A     "ONE_SEC_PULSE";
      JNB   _006;
      L     "08_LID_MECHANISM_DB".LID_2_VER_DN_OP_CUT_TIME;
      L     1;
      +I;
      T     "08_LID_MECHANISM_DB".LID_2_VER_DN_OP_CUT_TIME;
_006: NOP   0;
      A     L 0.0;
      A(;
      L     "08_LID_MECHANISM_DB".LID_2_VER_DN_OP_CUT_TIME;
      L     2;
      >=I;
      );
      =     "08_LID_MECHANISM_DB".LID_2_VER_DN_OP_CUT;
NETWORK
TITLE = LID LIFTER 2 VERTICAL DOWN ON INDICATION
      A     "ALWAYS_ON";
      A(;
      A     "08_LID_MECHANISM_DB".LID_LIFT_2_VER_DN_CMD;
      A     "HALF_SECOND_PULSE_TRAIN";
      O     "08_LID_MECHANISM_DB".LID_LIFT_2_VER_DN_LS;
      O     "MAIN_POWER_DB".LAMP_TEST_PB;
      );
      =     "08_LID_MECHANISM_DB".LID_LIFT_2_VER_DN_IND;
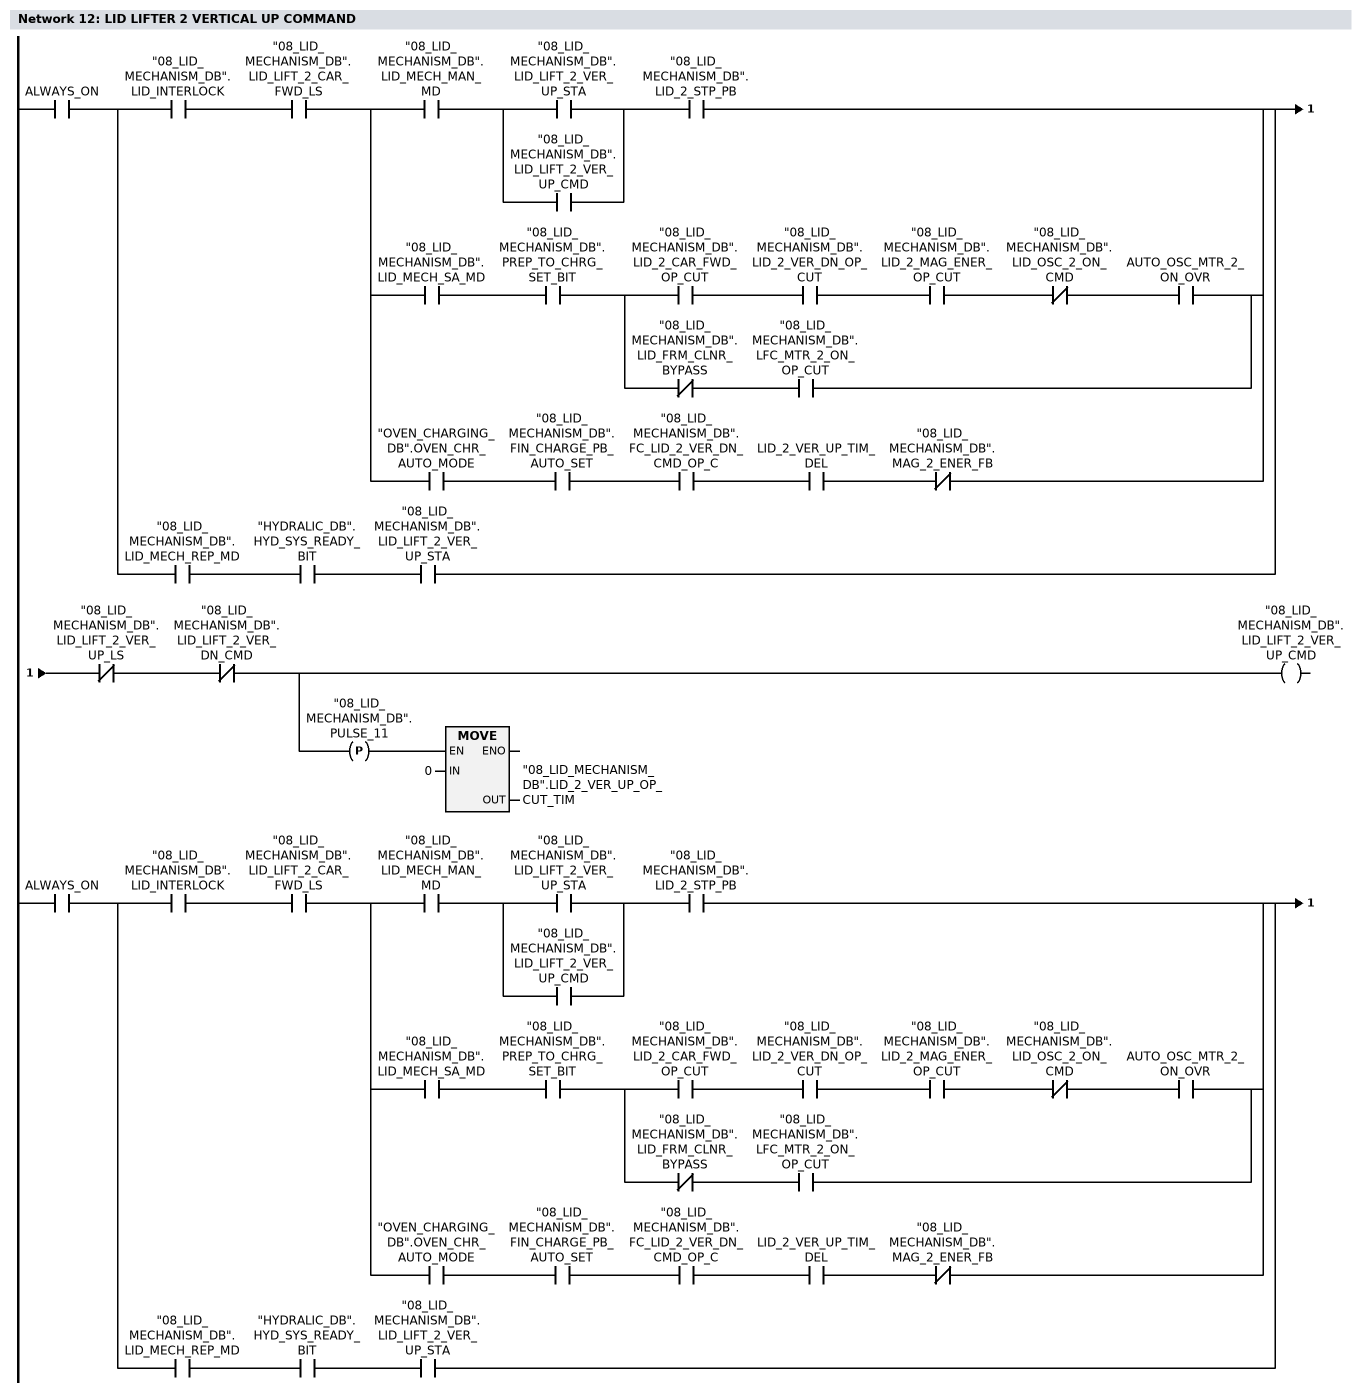
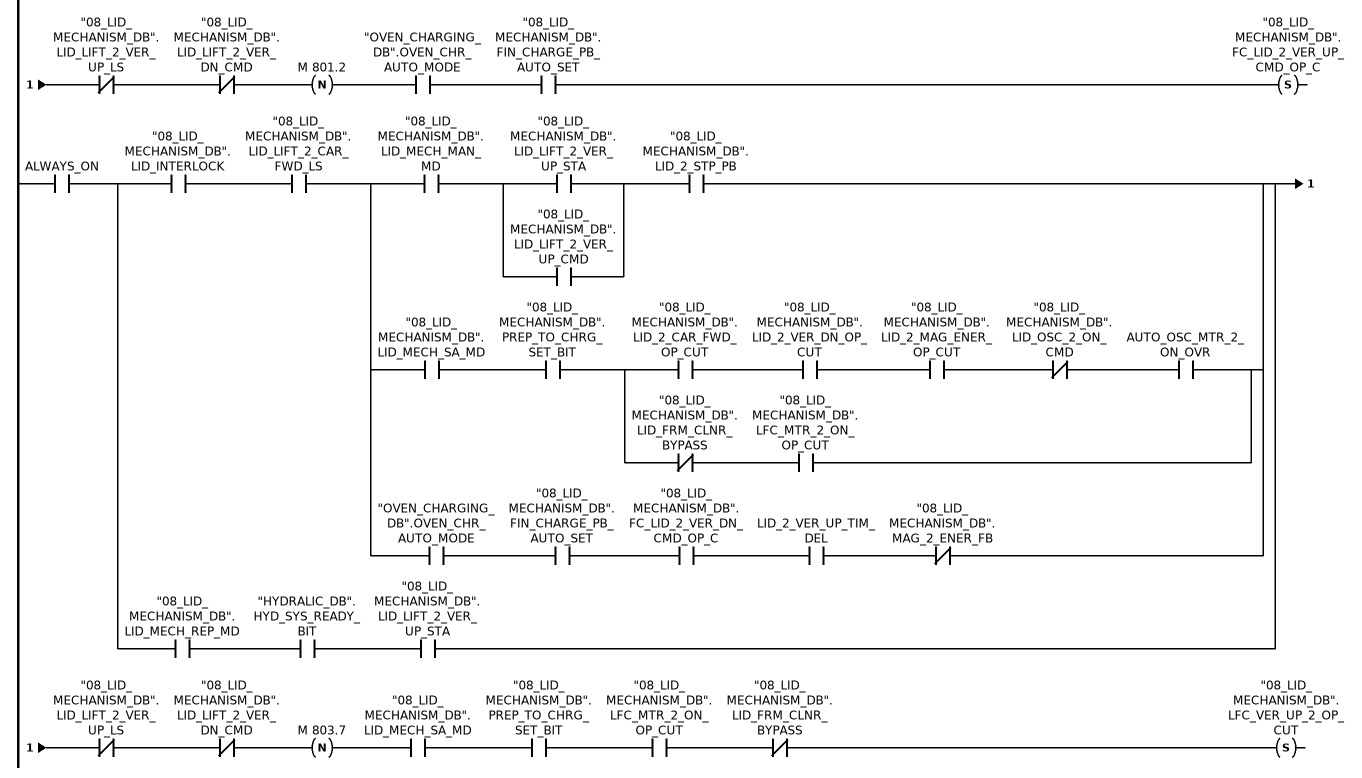
NETWORK
TITLE = LID LIFTER 2 VERTICAL UP COMMAND
      A     "ALWAYS_ON";
      A(;
      A     "08_LID_MECHANISM_DB".LID_INTERLOCK;
      A     "08_LID_MECHANISM_DB".LID_LIFT_2_CAR_FWD_LS;
      A(;
      A     "08_LID_MECHANISM_DB".LID_MECH_MAN_MD;
      A(;
      O     "08_LID_MECHANISM_DB".LID_LIFT_2_VER_UP_STA;
      O     "08_LID_MECHANISM_DB".LID_LIFT_2_VER_UP_CMD;
      );
      A     "08_LID_MECHANISM_DB".LID_2_STP_PB;
      O;
      A     "08_LID_MECHANISM_DB".LID_MECH_SA_MD;
      A     "08_LID_MECHANISM_DB".PREP_TO_CHRG_SET_BIT;
      A(;
      A     "08_LID_MECHANISM_DB".LID_2_CAR_FWD_OP_CUT;
      A     "08_LID_MECHANISM_DB".LID_2_VER_DN_OP_CUT;
      A     "08_LID_MECHANISM_DB".LID_2_MAG_ENER_OP_CUT;
      AN    "08_LID_MECHANISM_DB".LID_OSC_2_ON_CMD;
      A     "AUTO_OSC_MTR_2_ON_OVR";
      O;
      AN    "08_LID_MECHANISM_DB".LID_FRM_CLNR_BYPASS;
      A     "08_LID_MECHANISM_DB".LFC_MTR_2_ON_OP_CUT;
      );
      O;
      A     "OVEN_CHARGING_DB".OVEN_CHR_AUTO_MODE;
      A     "08_LID_MECHANISM_DB".FIN_CHARGE_PB_AUTO_SET;
      A     "08_LID_MECHANISM_DB".FC_LID_2_VER_DN_CMD_OP_C;
      A     "LID_2_VER_UP_TIM_DEL";
      AN    "08_LID_MECHANISM_DB".MAG_2_ENER_FB;
      );
      O;
      A     "08_LID_MECHANISM_DB".LID_MECH_REP_MD;
      A     "HYDRALIC_DB".HYD_SYS_READY_BIT;
      A     "08_LID_MECHANISM_DB".LID_LIFT_2_VER_UP_STA;
      );
      AN    "08_LID_MECHANISM_DB".LID_LIFT_2_VER_UP_LS;
      AN    "08_LID_MECHANISM_DB".LID_LIFT_2_VER_DN_CMD;
      =     L 0.0;
      A     L 0.0;
      BLD   102;
      =     "08_LID_MECHANISM_DB".LID_LIFT_2_VER_UP_CMD;
      A     L 0.0;
      FP    "08_LID_MECHANISM_DB".PULSE_11;
      JNB   _007;
      L     0;
      T     "08_LID_MECHANISM_DB".LID_2_VER_UP_OP_CUT_TIM;
_007: NOP   0;
      A(;
      A     L 0.0;
      FN    M 801.2;
      );
      A     "OVEN_CHARGING_DB".OVEN_CHR_AUTO_MODE;
      A     "08_LID_MECHANISM_DB".FIN_CHARGE_PB_AUTO_SET;
      S     "08_LID_MECHANISM_DB".FC_LID_2_VER_UP_CMD_OP_C;
      A(;
      A     L 0.0;
      FN    M 803.7;
      );
      A     "08_LID_MECHANISM_DB".LID_MECH_SA_MD;
      A     "08_LID_MECHANISM_DB".PREP_TO_CHRG_SET_BIT;
      A     "08_LID_MECHANISM_DB".LFC_MTR_2_ON_OP_CUT;
      AN    "08_LID_MECHANISM_DB".LID_FRM_CLNR_BYPASS;
      S     "08_LID_MECHANISM_DB".LFC_VER_UP_2_OP_CUT;
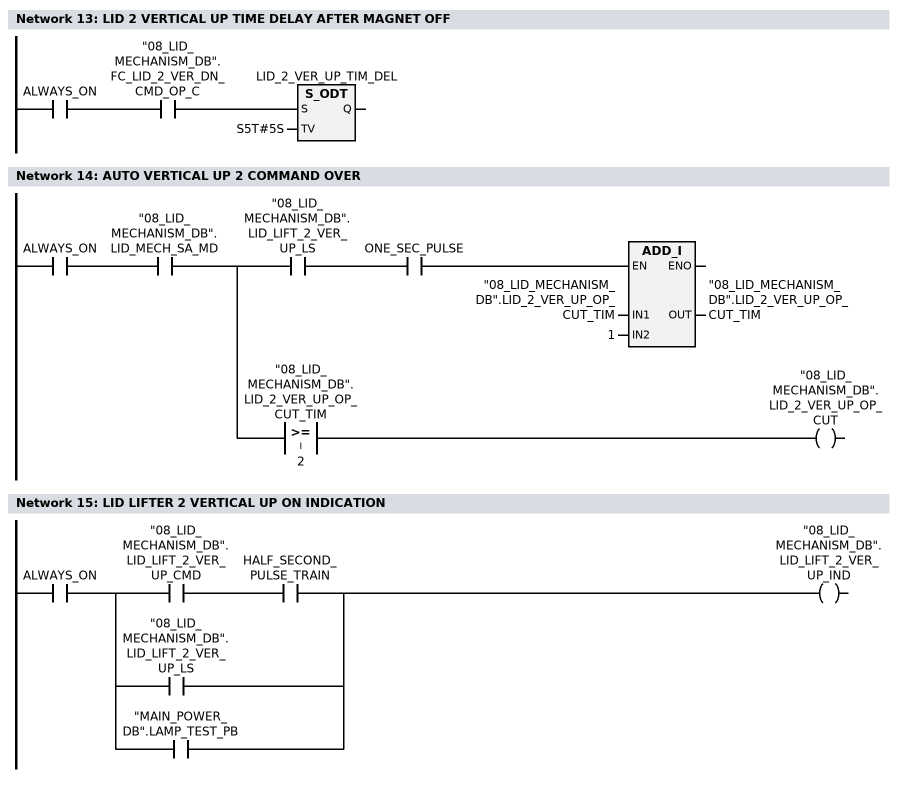
NETWORK
TITLE = LID 2 VERTICAL UP TIME DELAY AFTER MAGNET OFF
      A     "ALWAYS_ON";
      A     "08_LID_MECHANISM_DB".FC_LID_2_VER_DN_CMD_OP_C;
      L     S5T#5S;
      SD    "LID_2_VER_UP_TIM_DEL";
      NOP   0;
      NOP   0;
      NOP   0;
      NOP   0;
NETWORK
TITLE = AUTO VERTICAL UP 2 COMMAND OVER
      A     "ALWAYS_ON";
      A     "08_LID_MECHANISM_DB".LID_MECH_SA_MD;
      =     L 0.0;
      A     L 0.0;
      A     "08_LID_MECHANISM_DB".LID_LIFT_2_VER_UP_LS;
      A     "ONE_SEC_PULSE";
      JNB   _008;
      L     "08_LID_MECHANISM_DB".LID_2_VER_UP_OP_CUT_TIM;
      L     1;
      +I;
      T     "08_LID_MECHANISM_DB".LID_2_VER_UP_OP_CUT_TIM;
_008: NOP   0;
      A     L 0.0;
      A(;
      L     "08_LID_MECHANISM_DB".LID_2_VER_UP_OP_CUT_TIM;
      L     2;
      >=I;
      );
      =     "08_LID_MECHANISM_DB".LID_2_VER_UP_OP_CUT;
NETWORK
TITLE = LID LIFTER 2 VERTICAL UP ON INDICATION
      A     "ALWAYS_ON";
      A(;
      A     "08_LID_MECHANISM_DB".LID_LIFT_2_VER_UP_CMD;
      A     "HALF_SECOND_PULSE_TRAIN";
      O     "08_LID_MECHANISM_DB".LID_LIFT_2_VER_UP_LS;
      O     "MAIN_POWER_DB".LAMP_TEST_PB;
      );
      =     "08_LID_MECHANISM_DB".LID_LIFT_2_VER_UP_IND;
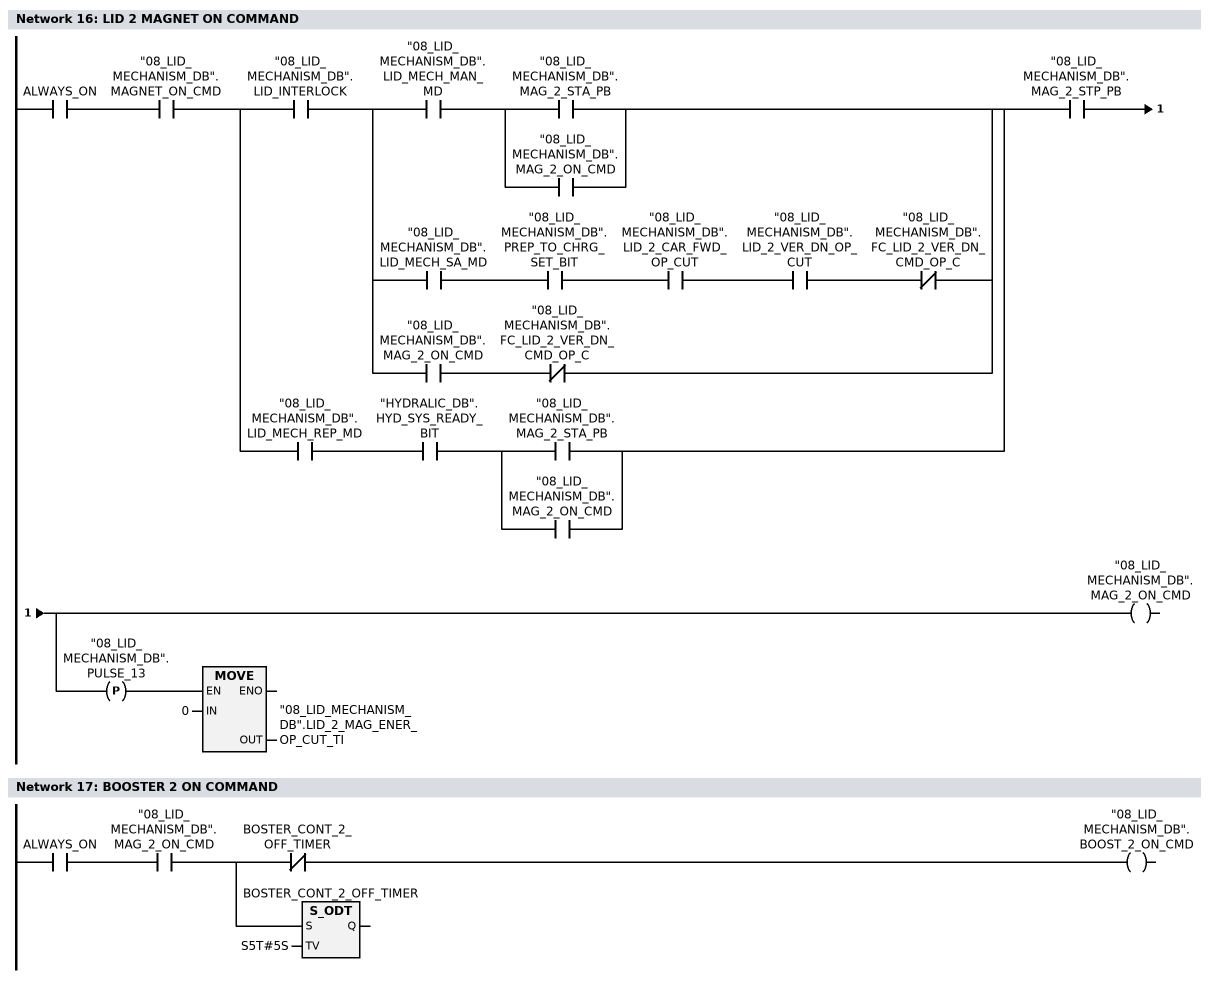
NETWORK
TITLE = LID 2 MAGNET ON COMMAND
      A     "ALWAYS_ON";
      A     "08_LID_MECHANISM_DB".MAGNET_ON_CMD;
      A(;
      A     "08_LID_MECHANISM_DB".LID_INTERLOCK;
      A(;
      A     "08_LID_MECHANISM_DB".LID_MECH_MAN_MD;
      A(;
      O     "08_LID_MECHANISM_DB".MAG_2_STA_PB;
      O     "08_LID_MECHANISM_DB".MAG_2_ON_CMD;
      );
      O;
      A     "08_LID_MECHANISM_DB".LID_MECH_SA_MD;
      A     "08_LID_MECHANISM_DB".PREP_TO_CHRG_SET_BIT;
      A     "08_LID_MECHANISM_DB".LID_2_CAR_FWD_OP_CUT;
      A     "08_LID_MECHANISM_DB".LID_2_VER_DN_OP_CUT;
      AN    "08_LID_MECHANISM_DB".FC_LID_2_VER_DN_CMD_OP_C;
      O;
      A     "08_LID_MECHANISM_DB".MAG_2_ON_CMD;
      AN    "08_LID_MECHANISM_DB".FC_LID_2_VER_DN_CMD_OP_C;
      );
      O;
      A     "08_LID_MECHANISM_DB".LID_MECH_REP_MD;
      A     "HYDRALIC_DB".HYD_SYS_READY_BIT;
      A(;
      O     "08_LID_MECHANISM_DB".MAG_2_STA_PB;
      O     "08_LID_MECHANISM_DB".MAG_2_ON_CMD;
      );
      );
      A     "08_LID_MECHANISM_DB".MAG_2_STP_PB;
      =     L 0.0;
      A     L 0.0;
      BLD   102;
      =     "08_LID_MECHANISM_DB".MAG_2_ON_CMD;
      A     L 0.0;
      FP    "08_LID_MECHANISM_DB".PULSE_13;
      JNB   _009;
      L     0;
      T     "08_LID_MECHANISM_DB".LID_2_MAG_ENER_OP_CUT_TI;
_009: NOP   0;
NETWORK
TITLE = BOOSTER 2 ON COMMAND
      A     "ALWAYS_ON";
      A     "08_LID_MECHANISM_DB".MAG_2_ON_CMD;
      =     L 0.0;
      A     L 0.0;
      AN    "BOSTER_CONT_2_OFF_TIMER";
      =     "08_LID_MECHANISM_DB".BOOST_2_ON_CMD;
      A     L 0.0;
      L     S5T#5S;
      SD    "BOSTER_CONT_2_OFF_TIMER";
      NOP   0;
      NOP   0;
      NOP   0;
      NOP   0;
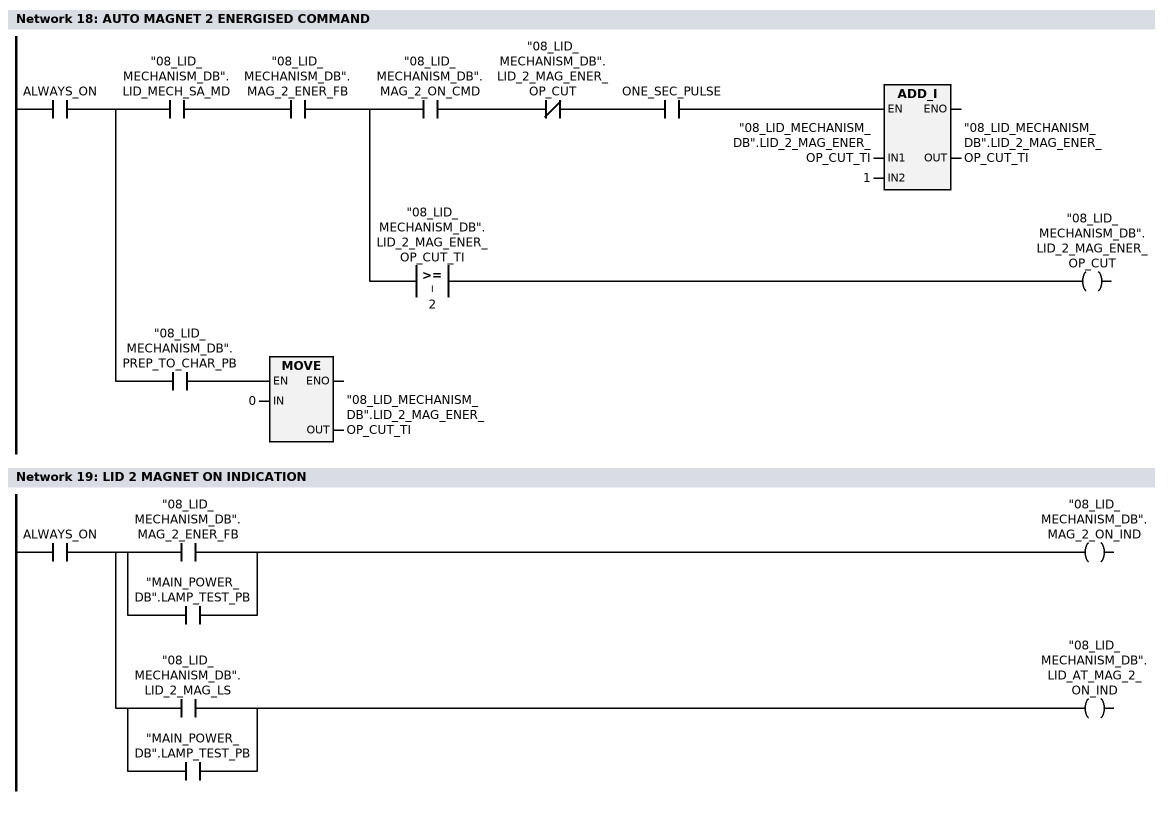
NETWORK
TITLE = AUTO MAGNET 2 ENERGISED COMMAND
      A     "ALWAYS_ON";
      =     L 0.0;
      A     L 0.0;
      A     "08_LID_MECHANISM_DB".LID_MECH_SA_MD;
      A     "08_LID_MECHANISM_DB".MAG_2_ENER_FB;
      =     L 0.1;
      A     L 0.1;
      A     "08_LID_MECHANISM_DB".MAG_2_ON_CMD;
      AN    "08_LID_MECHANISM_DB".LID_2_MAG_ENER_OP_CUT;
      A     "ONE_SEC_PULSE";
      JNB   _00a;
      L     "08_LID_MECHANISM_DB".LID_2_MAG_ENER_OP_CUT_TI;
      L     1;
      +I;
      T     "08_LID_MECHANISM_DB".LID_2_MAG_ENER_OP_CUT_TI;
_00a: NOP   0;
      A     L 0.1;
      A(;
      L     "08_LID_MECHANISM_DB".LID_2_MAG_ENER_OP_CUT_TI;
      L     2;
      >=I;
      );
      =     "08_LID_MECHANISM_DB".LID_2_MAG_ENER_OP_CUT;
      A     L 0.0;
      A     "08_LID_MECHANISM_DB".PREP_TO_CHAR_PB;
      JNB   _00b;
      L     0;
      T     "08_LID_MECHANISM_DB".LID_2_MAG_ENER_OP_CUT_TI;
_00b: NOP   0;
NETWORK
TITLE = LID 2 MAGNET ON INDICATION
      A     "ALWAYS_ON";
      =     L 0.0;
      A     L 0.0;
      A(;
      O     "08_LID_MECHANISM_DB".MAG_2_ENER_FB;
      O     "MAIN_POWER_DB".LAMP_TEST_PB;
      );
      =     "08_LID_MECHANISM_DB".MAG_2_ON_IND;
      A     L 0.0;
      A(;
      O     "08_LID_MECHANISM_DB".LID_2_MAG_LS;
      O     "MAIN_POWER_DB".LAMP_TEST_PB;
      );
      =     "08_LID_MECHANISM_DB".LID_AT_MAG_2_ON_IND;
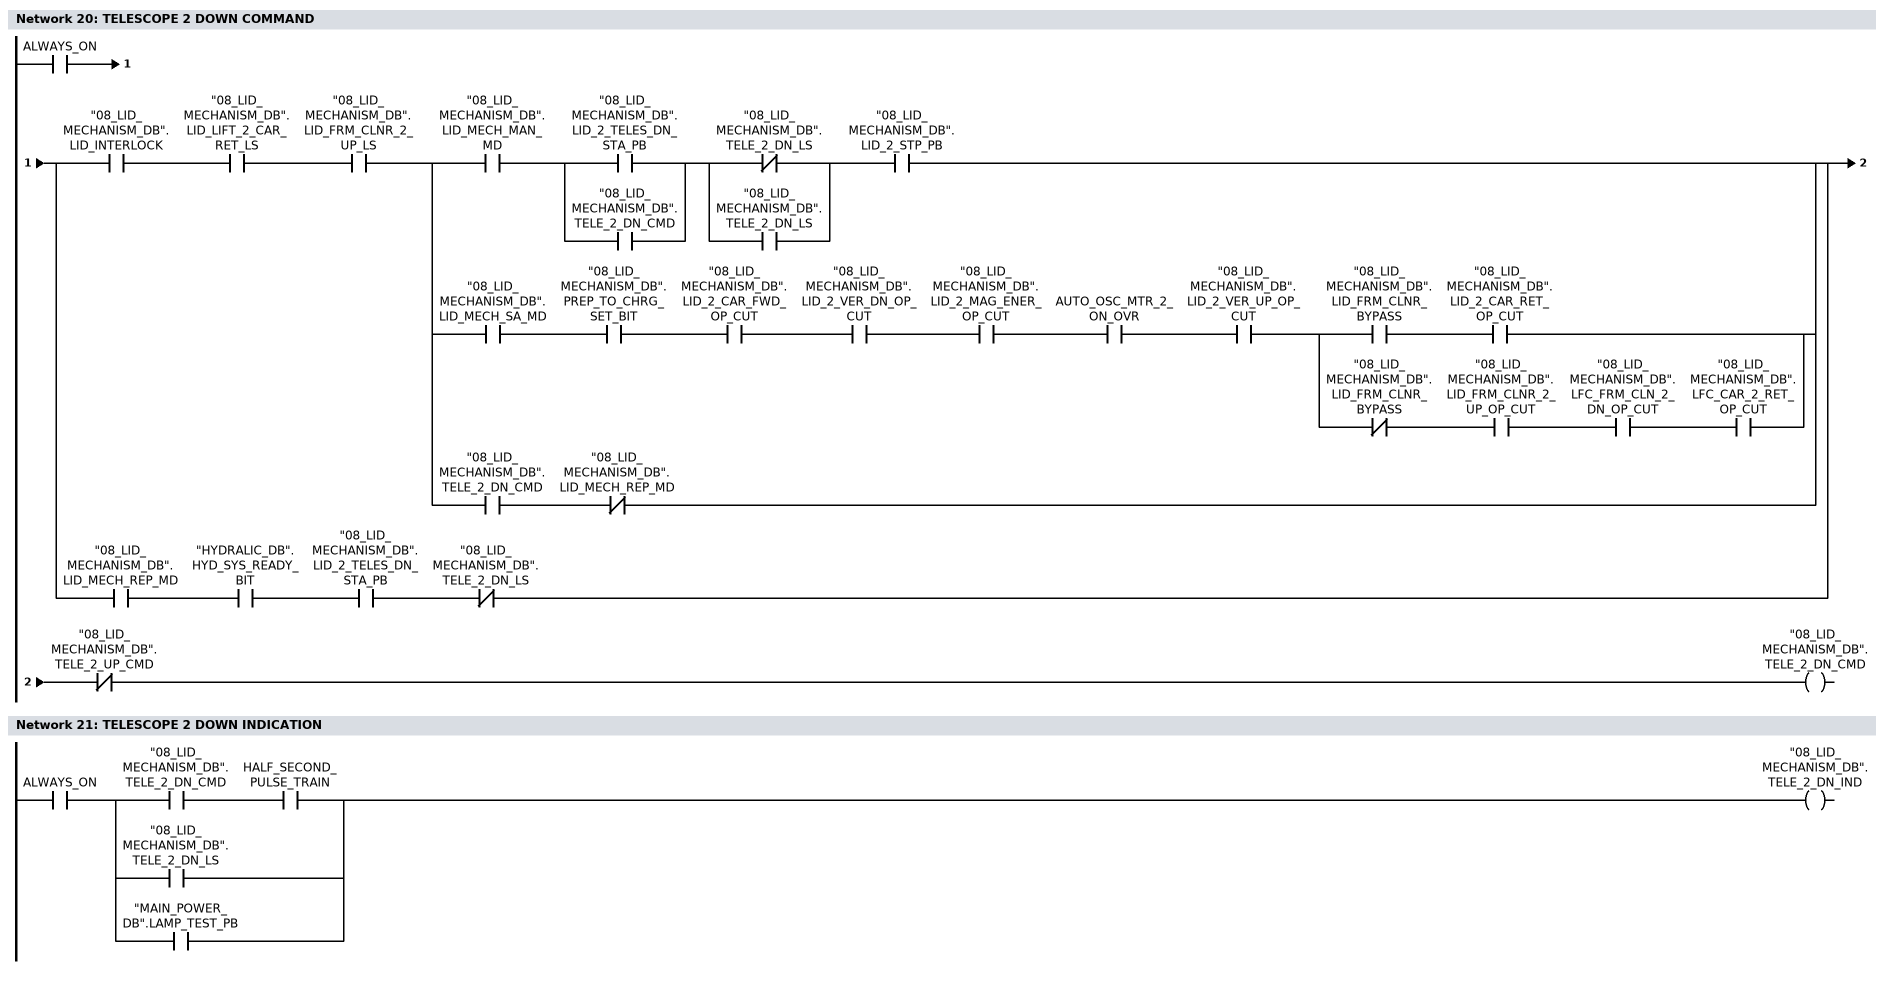
NETWORK
TITLE = TELESCOPE 2 DOWN COMMAND
      A     "ALWAYS_ON";
      A(;
      A     "08_LID_MECHANISM_DB".LID_INTERLOCK;
      A     "08_LID_MECHANISM_DB".LID_LIFT_2_CAR_RET_LS;
      A     "08_LID_MECHANISM_DB".LID_FRM_CLNR_2_UP_LS;
      A(;
      A     "08_LID_MECHANISM_DB".LID_MECH_MAN_MD;
      A(;
      O     "08_LID_MECHANISM_DB".LID_2_TELES_DN_STA_PB;
      O     "08_LID_MECHANISM_DB".TELE_2_DN_CMD;
      );
      A(;
      ON    "08_LID_MECHANISM_DB".TELE_2_DN_LS;
      O     "08_LID_MECHANISM_DB".TELE_2_DN_LS;
      );
      A     "08_LID_MECHANISM_DB".LID_2_STP_PB;
      O;
      A     "08_LID_MECHANISM_DB".LID_MECH_SA_MD;
      A     "08_LID_MECHANISM_DB".PREP_TO_CHRG_SET_BIT;
      A     "08_LID_MECHANISM_DB".LID_2_CAR_FWD_OP_CUT;
      A     "08_LID_MECHANISM_DB".LID_2_VER_DN_OP_CUT;
      A     "08_LID_MECHANISM_DB".LID_2_MAG_ENER_OP_CUT;
      A     "AUTO_OSC_MTR_2_ON_OVR";
      A     "08_LID_MECHANISM_DB".LID_2_VER_UP_OP_CUT;
      A(;
      A     "08_LID_MECHANISM_DB".LID_FRM_CLNR_BYPASS;
      A     "08_LID_MECHANISM_DB".LID_2_CAR_RET_OP_CUT;
      O;
      AN    "08_LID_MECHANISM_DB".LID_FRM_CLNR_BYPASS;
      A     "08_LID_MECHANISM_DB".LID_FRM_CLNR_2_UP_OP_CUT;
      A     "08_LID_MECHANISM_DB".LFC_FRM_CLN_2_DN_OP_CUT;
      A     "08_LID_MECHANISM_DB".LFC_CAR_2_RET_OP_CUT;
      );
      O;
      A     "08_LID_MECHANISM_DB".TELE_2_DN_CMD;
      AN    "08_LID_MECHANISM_DB".LID_MECH_REP_MD;
      );
      O;
      A     "08_LID_MECHANISM_DB".LID_MECH_REP_MD;
      A     "HYDRALIC_DB".HYD_SYS_READY_BIT;
      A     "08_LID_MECHANISM_DB".LID_2_TELES_DN_STA_PB;
      AN    "08_LID_MECHANISM_DB".TELE_2_DN_LS;
      );
      AN    "08_LID_MECHANISM_DB".TELE_2_UP_CMD;
      =     "08_LID_MECHANISM_DB".TELE_2_DN_CMD;
NETWORK
TITLE = TELESCOPE 2 DOWN INDICATION
      A     "ALWAYS_ON";
      A(;
      A     "08_LID_MECHANISM_DB".TELE_2_DN_CMD;
      A     "HALF_SECOND_PULSE_TRAIN";
      O     "08_LID_MECHANISM_DB".TELE_2_DN_LS;
      O     "MAIN_POWER_DB".LAMP_TEST_PB;
      );
      =     "08_LID_MECHANISM_DB".TELE_2_DN_IND;
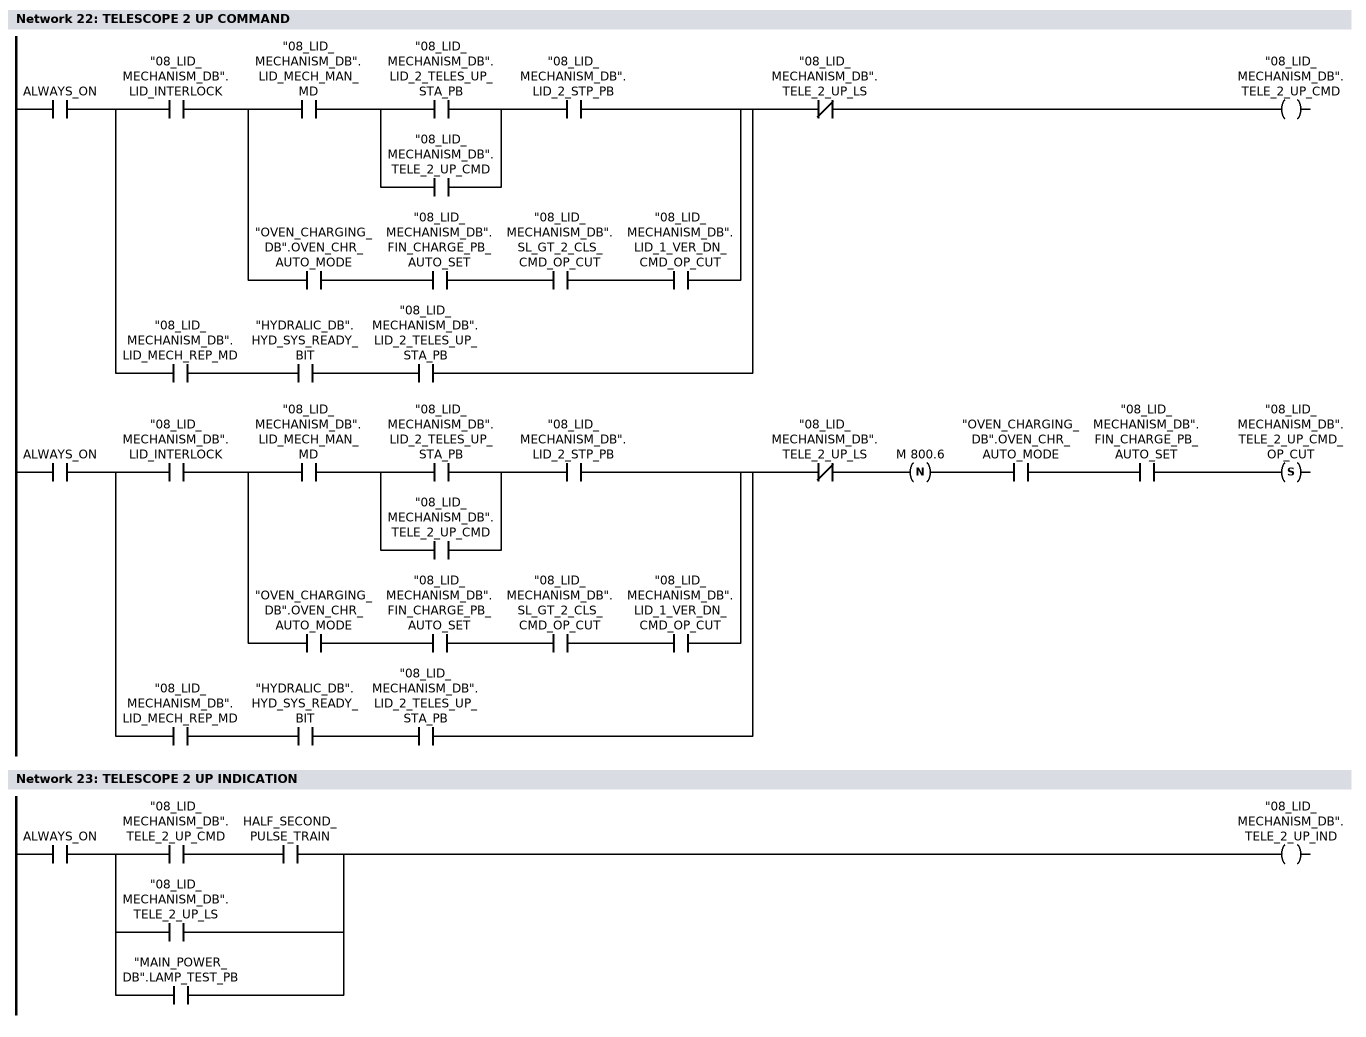
NETWORK
TITLE = TELESCOPE 2 UP COMMAND
      A     "ALWAYS_ON";
      A(;
      A     "08_LID_MECHANISM_DB".LID_INTERLOCK;
      A(;
      A     "08_LID_MECHANISM_DB".LID_MECH_MAN_MD;
      A(;
      O     "08_LID_MECHANISM_DB".LID_2_TELES_UP_STA_PB;
      O     "08_LID_MECHANISM_DB".TELE_2_UP_CMD;
      );
      A     "08_LID_MECHANISM_DB".LID_2_STP_PB;
      O;
      A     "OVEN_CHARGING_DB".OVEN_CHR_AUTO_MODE;
      A     "08_LID_MECHANISM_DB".FIN_CHARGE_PB_AUTO_SET;
      A     "08_LID_MECHANISM_DB".SL_GT_2_CLS_CMD_OP_CUT;
      A     "08_LID_MECHANISM_DB".LID_1_VER_DN_CMD_OP_CUT;
      );
      O;
      A     "08_LID_MECHANISM_DB".LID_MECH_REP_MD;
      A     "HYDRALIC_DB".HYD_SYS_READY_BIT;
      A     "08_LID_MECHANISM_DB".LID_2_TELES_UP_STA_PB;
      );
      AN    "08_LID_MECHANISM_DB".TELE_2_UP_LS;
      =     L 0.0;
      A     L 0.0;
      BLD   102;
      =     "08_LID_MECHANISM_DB".TELE_2_UP_CMD;
      A(;
      A     L 0.0;
      FN    M 800.6;
      );
      A     "OVEN_CHARGING_DB".OVEN_CHR_AUTO_MODE;
      A     "08_LID_MECHANISM_DB".FIN_CHARGE_PB_AUTO_SET;
      S     "08_LID_MECHANISM_DB".TELE_2_UP_CMD_OP_CUT;
NETWORK
TITLE = TELESCOPE 2 UP INDICATION
      A     "ALWAYS_ON";
      A(;
      A     "08_LID_MECHANISM_DB".TELE_2_UP_CMD;
      A     "HALF_SECOND_PULSE_TRAIN";
      O     "08_LID_MECHANISM_DB".TELE_2_UP_LS;
      O     "MAIN_POWER_DB".LAMP_TEST_PB;
      );
      =     "08_LID_MECHANISM_DB".TELE_2_UP_IND;
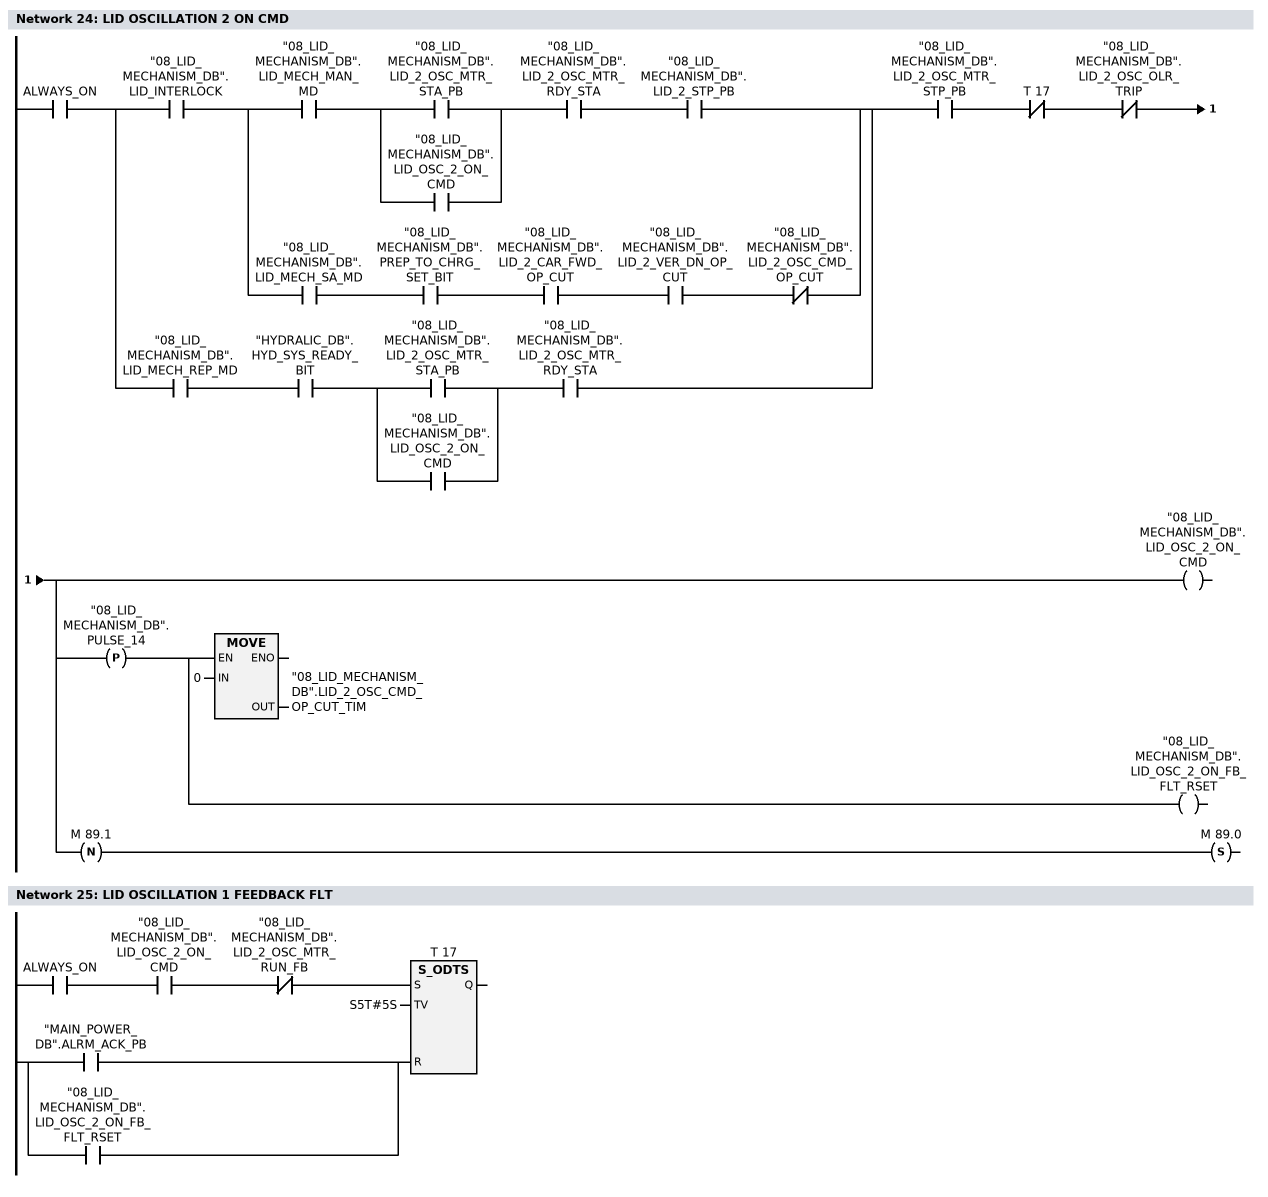
NETWORK
TITLE = LID OSCILLATION 2 ON CMD
      A     "ALWAYS_ON";
      A(;
      A     "08_LID_MECHANISM_DB".LID_INTERLOCK;
      A(;
      A     "08_LID_MECHANISM_DB".LID_MECH_MAN_MD;
      A(;
      O     "08_LID_MECHANISM_DB".LID_2_OSC_MTR_STA_PB;
      O     "08_LID_MECHANISM_DB".LID_OSC_2_ON_CMD;
      );
      A     "08_LID_MECHANISM_DB".LID_2_OSC_MTR_RDY_STA;
      A     "08_LID_MECHANISM_DB".LID_2_STP_PB;
      O;
      A     "08_LID_MECHANISM_DB".LID_MECH_SA_MD;
      A     "08_LID_MECHANISM_DB".PREP_TO_CHRG_SET_BIT;
      A     "08_LID_MECHANISM_DB".LID_2_CAR_FWD_OP_CUT;
      A     "08_LID_MECHANISM_DB".LID_2_VER_DN_OP_CUT;
      AN    "08_LID_MECHANISM_DB".LID_2_OSC_CMD_OP_CUT;
      );
      O;
      A     "08_LID_MECHANISM_DB".LID_MECH_REP_MD;
      A     "HYDRALIC_DB".HYD_SYS_READY_BIT;
      A(;
      O     "08_LID_MECHANISM_DB".LID_2_OSC_MTR_STA_PB;
      O     "08_LID_MECHANISM_DB".LID_OSC_2_ON_CMD;
      );
      A     "08_LID_MECHANISM_DB".LID_2_OSC_MTR_RDY_STA;
      );
      A     "08_LID_MECHANISM_DB".LID_2_OSC_MTR_STP_PB;
      AN    T 17;
      AN    "08_LID_MECHANISM_DB".LID_2_OSC_OLR_TRIP;
      =     L 0.0;
      A     L 0.0;
      BLD   102;
      =     "08_LID_MECHANISM_DB".LID_OSC_2_ON_CMD;
      A     L 0.0;
      FP    "08_LID_MECHANISM_DB".PULSE_14;
      =     L 0.1;
      A     L 0.1;
      JNB   _00c;
      L     0;
      T     "08_LID_MECHANISM_DB".LID_2_OSC_CMD_OP_CUT_TIM;
_00c: NOP   0;
      A     L 0.1;
      BLD   102;
      =     "08_LID_MECHANISM_DB".LID_OSC_2_ON_FB_FLT_RSET;
      A     L 0.0;
      FN    M 89.1;
      S     M 89.0;
NETWORK
TITLE = LID OSCILLATION 1 FEEDBACK FLT
      A     "ALWAYS_ON";
      A     "08_LID_MECHANISM_DB".LID_OSC_2_ON_CMD;
      AN    "08_LID_MECHANISM_DB".LID_2_OSC_MTR_RUN_FB;
      L     S5T#5S;
      SS    T 17;
      A(;
      O     "MAIN_POWER_DB".ALRM_ACK_PB;
      O     "08_LID_MECHANISM_DB".LID_OSC_2_ON_FB_FLT_RSET;
      );
      R     T 17;
      NOP   0;
      NOP   0;
      NOP   0;
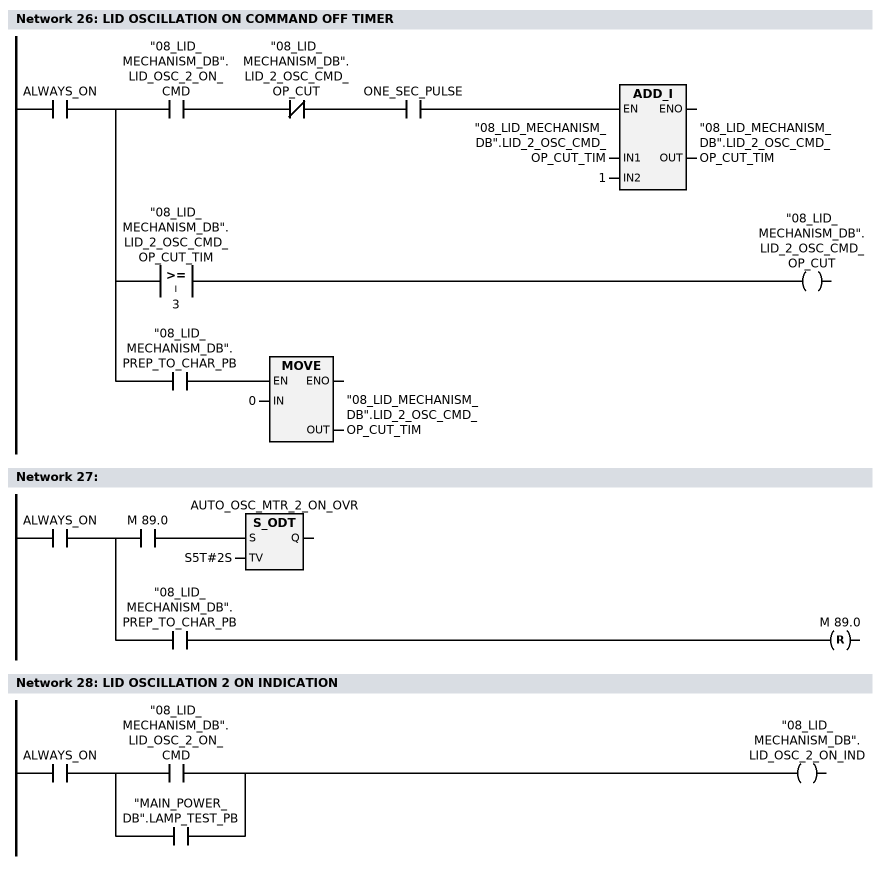
NETWORK
TITLE = LID OSCILLATION ON COMMAND OFF TIMER
      A     "ALWAYS_ON";
      =     L 0.0;
      A     L 0.0;
      A     "08_LID_MECHANISM_DB".LID_OSC_2_ON_CMD;
      AN    "08_LID_MECHANISM_DB".LID_2_OSC_CMD_OP_CUT;
      A     "ONE_SEC_PULSE";
      JNB   _00d;
      L     "08_LID_MECHANISM_DB".LID_2_OSC_CMD_OP_CUT_TIM;
      L     1;
      +I;
      T     "08_LID_MECHANISM_DB".LID_2_OSC_CMD_OP_CUT_TIM;
_00d: NOP   0;
      A     L 0.0;
      A(;
      L     "08_LID_MECHANISM_DB".LID_2_OSC_CMD_OP_CUT_TIM;
      L     3;
      >=I;
      );
      =     "08_LID_MECHANISM_DB".LID_2_OSC_CMD_OP_CUT;
      A     L 0.0;
      A     "08_LID_MECHANISM_DB".PREP_TO_CHAR_PB;
      JNB   _00e;
      L     0;
      T     "08_LID_MECHANISM_DB".LID_2_OSC_CMD_OP_CUT_TIM;
_00e: NOP   0;
NETWORK
TITLE =
      A     "ALWAYS_ON";
      =     L 0.0;
      A     L 0.0;
      A     M 89.0;
      L     S5T#2S;
      SD    "AUTO_OSC_MTR_2_ON_OVR";
      NOP   0;
      NOP   0;
      NOP   0;
      NOP   0;
      A     L 0.0;
      A     "08_LID_MECHANISM_DB".PREP_TO_CHAR_PB;
      R     M 89.0;
NETWORK
TITLE = LID OSCILLATION 2 ON INDICATION
//CHECK IT
      A     "ALWAYS_ON";
      A(;
      O     "08_LID_MECHANISM_DB".LID_OSC_2_ON_CMD;
      O     "MAIN_POWER_DB".LAMP_TEST_PB;
      );
      =     "08_LID_MECHANISM_DB".LID_OSC_2_ON_IND;
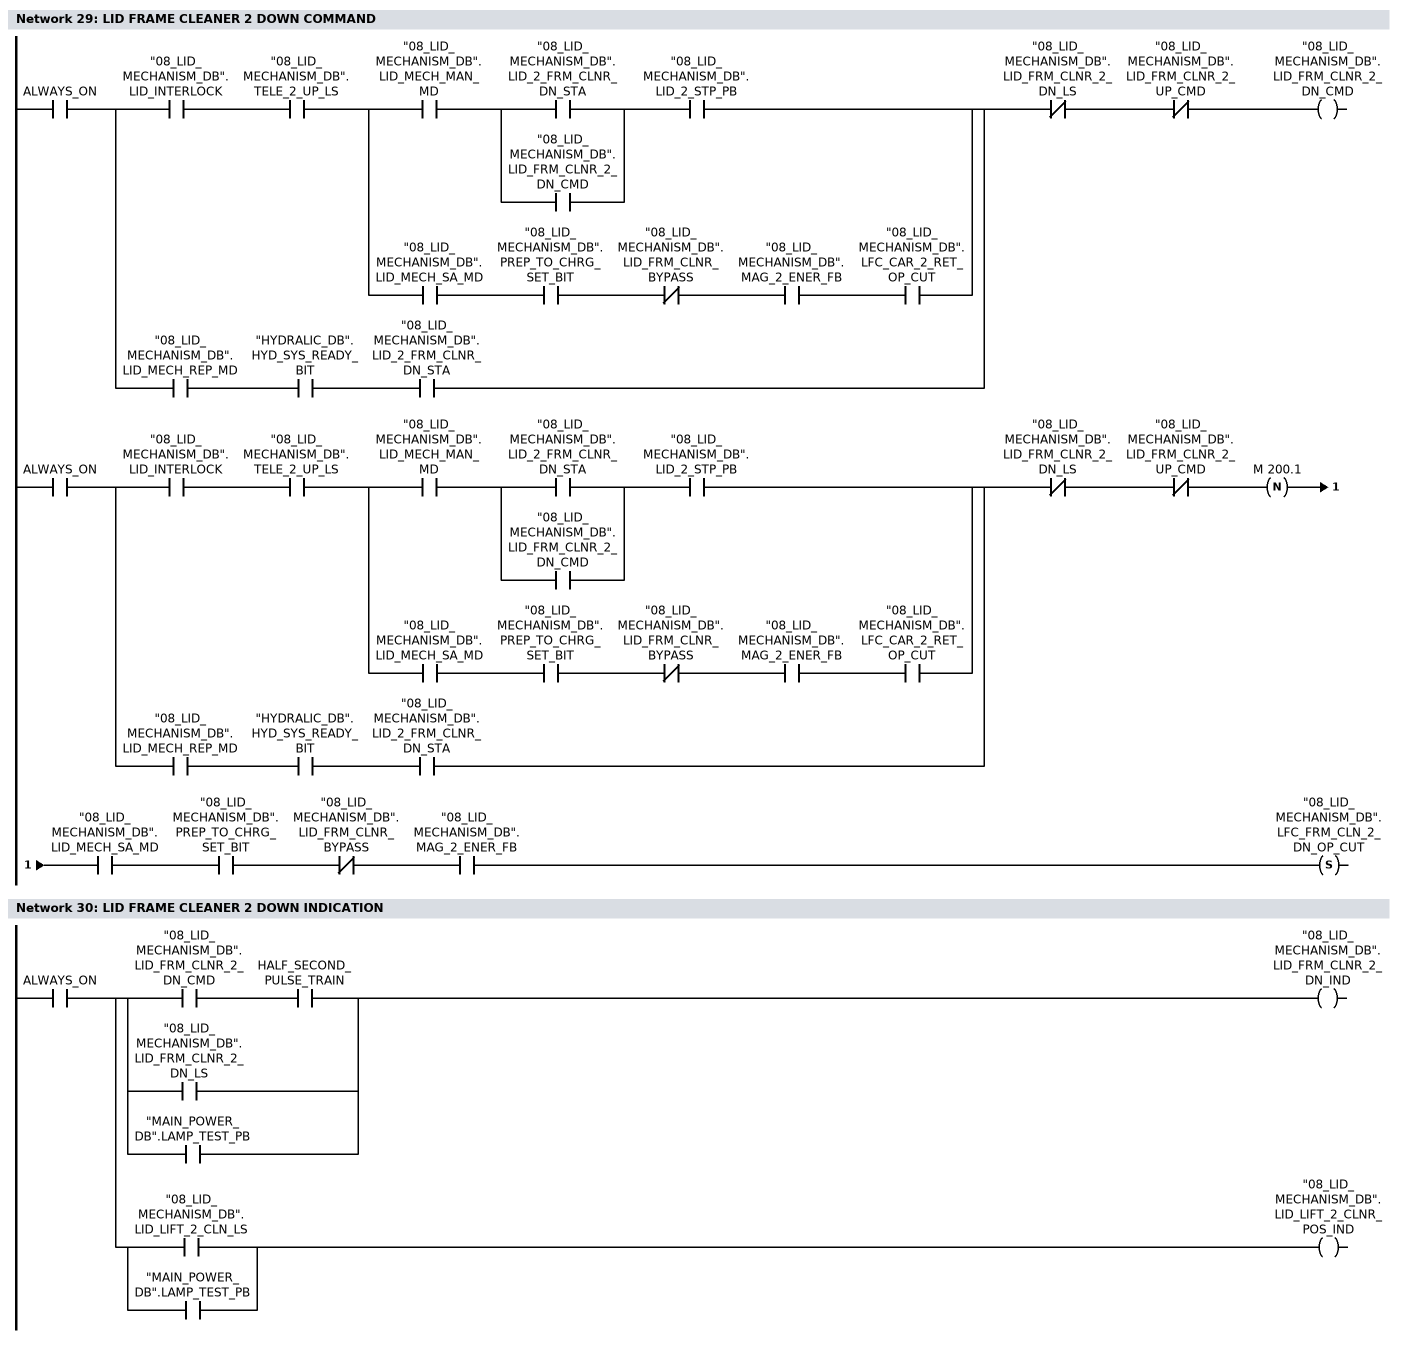
NETWORK
TITLE = LID FRAME CLEANER 2 DOWN COMMAND
      A     "ALWAYS_ON";
      A(;
      A     "08_LID_MECHANISM_DB".LID_INTERLOCK;
      A     "08_LID_MECHANISM_DB".TELE_2_UP_LS;
      A(;
      A     "08_LID_MECHANISM_DB".LID_MECH_MAN_MD;
      A(;
      O     "08_LID_MECHANISM_DB".LID_2_FRM_CLNR_DN_STA;
      O     "08_LID_MECHANISM_DB".LID_FRM_CLNR_2_DN_CMD;
      );
      A     "08_LID_MECHANISM_DB".LID_2_STP_PB;
      O;
      A     "08_LID_MECHANISM_DB".LID_MECH_SA_MD;
      A     "08_LID_MECHANISM_DB".PREP_TO_CHRG_SET_BIT;
      AN    "08_LID_MECHANISM_DB".LID_FRM_CLNR_BYPASS;
      A     "08_LID_MECHANISM_DB".MAG_2_ENER_FB;
      A     "08_LID_MECHANISM_DB".LFC_CAR_2_RET_OP_CUT;
      );
      O;
      A     "08_LID_MECHANISM_DB".LID_MECH_REP_MD;
      A     "HYDRALIC_DB".HYD_SYS_READY_BIT;
      A     "08_LID_MECHANISM_DB".LID_2_FRM_CLNR_DN_STA;
      );
      AN    "08_LID_MECHANISM_DB".LID_FRM_CLNR_2_DN_LS;
      AN    "08_LID_MECHANISM_DB".LID_FRM_CLNR_2_UP_CMD;
      =     L 0.0;
      A     L 0.0;
      BLD   102;
      =     "08_LID_MECHANISM_DB".LID_FRM_CLNR_2_DN_CMD;
      A(;
      A     L 0.0;
      FN    M 200.1;
      );
      A     "08_LID_MECHANISM_DB".LID_MECH_SA_MD;
      A     "08_LID_MECHANISM_DB".PREP_TO_CHRG_SET_BIT;
      AN    "08_LID_MECHANISM_DB".LID_FRM_CLNR_BYPASS;
      A     "08_LID_MECHANISM_DB".MAG_2_ENER_FB;
      S     "08_LID_MECHANISM_DB".LFC_FRM_CLN_2_DN_OP_CUT;
NETWORK
TITLE = LID FRAME CLEANER 2 DOWN INDICATION
      A     "ALWAYS_ON";
      =     L 0.0;
      A     L 0.0;
      A(;
      A     "08_LID_MECHANISM_DB".LID_FRM_CLNR_2_DN_CMD;
      A     "HALF_SECOND_PULSE_TRAIN";
      O     "08_LID_MECHANISM_DB".LID_FRM_CLNR_2_DN_LS;
      O     "MAIN_POWER_DB".LAMP_TEST_PB;
      );
      =     "08_LID_MECHANISM_DB".LID_FRM_CLNR_2_DN_IND;
      A     L 0.0;
      A(;
      O     "08_LID_MECHANISM_DB".LID_LIFT_2_CLN_LS;
      O     "MAIN_POWER_DB".LAMP_TEST_PB;
      );
      =     "08_LID_MECHANISM_DB".LID_LIFT_2_CLNR_POS_IND;
